LIN {X 0,Y 572.946,Z 406.186,A -85,B 0,C 180,E1 -2251.405,E2 -2251.405} C_VEL
LIN {X 0,Y 572.959,Z 403.811,A -85,B 0,C 180,E1 -2252.812,E2 -2252.812} C_VEL
LIN {X 0,Y 573.014,Z 400.897,A -85,B 0,C 180,E1 -2253.868,E2 -2253.868} C_VEL
LIN {X 0,Y 572.963,Z 396.95,A -85,B 0,C 180,E1 -2254.925,E2 -2254.925} C_VEL
LIN {X 0,Y 573.093,Z 391.869,A -85,B 0,C 180,E1 -2255.983,E2 -2255.983} C_VEL
LIN {X 0,Y 573.103,Z 385.471,A -85,B 0,C 180,E1 -2257.043,E2 -2257.043} C_VEL
LIN {X 0,Y 573.177,Z 377.482,A -85,B 0,C 180,E1 -2258.106,E2 -2258.106} C_VEL
LIN {X 0,Y 573.253,Z 369.34,A -85,B 0,C 180,E1 -2258.992,E2 -2258.992} C_VEL
LIN {X 0,Y 573.349,Z 359.406,A -85,B 0,C 180,E1 -2259.881,E2 -2259.881} C_VEL
LIN {X 0,Y 573.523,Z 348.194,A -85,B 0,C 180,E1 -2260.68,E2 -2260.68} C_VEL
LIN {X 0,Y 573.627,Z 337.186,A -85,B 0,C 180,E1 -2261.304,E2 -2261.304} C_VEL
LIN {X 0,Y 573.705,Z 324.996,A -85,B 0,C 180,E1 -2261.84,E2 -2261.84} C_VEL
LIN {X 0,Y 573.851,Z 312.2,A -85,B 0,C 180,E1 -2262.241,E2 -2262.241} C_VEL
LIN {X 0,Y 573.908,Z 298.642,A -85,B 0,C 180,E1 -2262.509,E2 -2262.509} C_VEL
LIN {X 0,Y 573.923,Z 199.106,A -85,B 0,C 180,E1 -2263.765,E2 -2263.765} C_VEL
LIN {X 0,Y 573.375,Z 195.407,A -85,B 0,C 180,E1 -2263.85,E2 -2263.85} C_VEL
LIN {X 0,Y 573.472,Z 178.674,A -85,B 0,C 180,E1 -2266.371,E2 -2266.371} C_VEL
LIN {X 0,Y 573.665,Z 161.996,A -85,B 0,C 180,E1 -2268.944,E2 -2268.944} C_VEL
LIN {X 0,Y 573.818,Z 145.276,A -85,B 0,C 180,E1 -2271.557,E2 -2271.557} C_VEL
LIN {X 0,Y 573.241,Z 142.129,A -85,B 0,C 180,E1 -2272.123,E2 -2272.123} C_VEL
LIN {X 0,Y 573.219,Z 142.079,A -85,B 0,C 180,E1 -2274.867,E2 -2274.867} C_VEL
LIN {X 0,Y 573.259,Z 142.075,A -85,B 0,C 180,E1 -2277.765,E2 -2277.765} C_VEL
LIN {X 0,Y 573.227,Z 142.075,A -85,B 0,C 180,E1 -2280.176,E2 -2280.176} C_VEL
LIN {X 0,Y 573.246,Z 142.076,A -85,B 0,C 180,E1 -2282.644,E2 -2282.644} C_VEL
LIN {X 0,Y 573.2,Z 142.088,A -85,B 0,C 180,E1 -2285.187,E2 -2285.187} C_VEL
LIN {X 0,Y 573.223,Z 142.075,A -85,B 0,C 180,E1 -2287.807,E2 -2287.807} C_VEL
LIN {X 0,Y 573.238,Z 142.076,A -85,B 0,C 180,E1 -2290.524,E2 -2290.524} C_VEL
LIN {X 0,Y 573.229,Z 142.077,A -85,B 0,C 180,E1 -2293.667,E2 -2293.667} C_VEL
LIN {X 0,Y 573.223,Z 142.079,A -85,B 0,C 180,E1 -2296.639,E2 -2296.639} C_VEL
LIN {X 0,Y 573.236,Z 142.078,A -85,B 0,C 180,E1 -2299.474,E2 -2299.474} C_VEL
LIN {X 0,Y 573.224,Z 142.074,A -85,B 0,C 180,E1 -2302.191,E2 -2302.191} C_VEL
LIN {X 0,Y 573.23,Z 142.08,A -85,B 0,C 180,E1 -2305.227,E2 -2305.227} C_VEL
LIN {X 0,Y 573.227,Z 142.076,A -85,B 0,C 180,E1 -2308.184,E2 -2308.184} C_VEL
LIN {X 0,Y 573.246,Z 142.078,A -85,B 0,C 180,E1 -2310.633,E2 -2310.633} C_VEL
LIN {X 0,Y 573.238,Z 142.082,A -85,B 0,C 180,E1 -2313.023,E2 -2313.023} C_VEL
LIN {X 0,Y 573.26,Z 142.072,A -85,B 0,C 180,E1 -2315.365,E2 -2315.365} C_VEL
LIN {X 0,Y 573.215,Z 142.081,A -85,B 0,C 180,E1 -2318.419,E2 -2318.419} C_VEL
LIN {X 0,Y 573.265,Z 142.08,A -85,B 0,C 180,E1 -2320.728,E2 -2320.728} C_VEL
LIN {X 0,Y 573.234,Z 142.074,A -85,B 0,C 180,E1 -2323.621,E2 -2323.621} C_VEL
LIN {X 0,Y 573.251,Z 142.073,A -85,B 0,C 180,E1 -2325.806,E2 -2325.806} C_VEL
LIN {X 0,Y 573.277,Z 142.077,A -85,B 0,C 180,E1 -2328.731,E2 -2328.731} C_VEL
LIN {X 0,Y 573.239,Z 142.074,A -85,B 0,C 180,E1 -2331.54,E2 -2331.54} C_VEL
LIN {X 0,Y 573.219,Z 142.076,A -85,B 0,C 180,E1 -2333.665,E2 -2333.665} C_VEL
LIN {X 0,Y 573.201,Z 142.077,A -85,B 0,C 180,E1 -2335.781,E2 -2335.781} C_VEL
LIN {X 0,Y 573.284,Z 142.07,A -85,B 0,C 180,E1 -2337.892,E2 -2337.892} C_VEL
LIN {X 0,Y 573.329,Z 142.068,A -85,B 0,C 180,E1 -2340.702,E2 -2340.702} C_VEL
LIN {X 0,Y 573.215,Z 142.076,A -85,B 0,C 180,E1 -2343.515,E2 -2343.515} C_VEL
LIN {X 0,Y 573.27,Z 142.07,A -85,B 0,C 180,E1 -2345.628,E2 -2345.628} C_VEL
LIN {X 0,Y 573.275,Z 142.077,A -85,B 0,C 180,E1 -2348.46,E2 -2348.46} C_VEL
LIN {X 0,Y 573.265,Z 142.07,A -85,B 0,C 180,E1 -2351.312,E2 -2351.312} C_VEL
LIN {X 0,Y 573.267,Z 142.078,A -85,B 0,C 180,E1 -2354.425,E2 -2354.425} C_VEL
LIN {X 0,Y 573.246,Z 142.073,A -85,B 0,C 180,E1 -2357.112,E2 -2357.112} C_VEL
LIN {X 0,Y 573.244,Z 142.081,A -85,B 0,C 180,E1 -2360.077,E2 -2360.077} C_VEL
LIN {X 0,Y 573.236,Z 142.082,A -85,B 0,C 180,E1 -2362.338,E2 -2362.338} C_VEL
LIN {X 0,Y 573.239,Z 142.076,A -85,B 0,C 180,E1 -2364.409,E2 -2364.409} C_VEL
LIN {X 0,Y 572.612,Z 142.157,A -85,B 0,C 180,E1 -2364.995,E2 -2364.995} C_VEL
LIN {X 0,Y 569.767,Z 142.513,A -85,B 0,C 180,E1 -2365.947,E2 -2365.947} C_VEL
LIN {X 0,Y 567.337,Z 142.81,A -85,B 0,C 180,E1 -2366.713,E2 -2366.713} C_VEL
LIN {X 0,Y 566.287,Z 142.939,A -85,B 0,C 180,E1 -2367.304,E2 -2367.304} C_VEL
LIN {X 0,Y 566.2,Z 142.951,A -85,B 0,C 180,E1 -2367.504,E2 -2367.504} C_VEL
LIN {X 0,Y 566.194,Z 142.956,A -85,B 0,C 180,E1 -2369.769,E2 -2369.769} C_VEL
LIN {X 0,Y 566.195,Z 142.954,A -85,B 0,C 180,E1 -2372.431,E2 -2372.431} C_VEL
LIN {X 0,Y 566.192,Z 142.946,A -85,B 0,C 180,E1 -2374.994,E2 -2374.994} C_VEL
LIN {X 0,Y 566.188,Z 142.952,A -85,B 0,C 180,E1 -2377.462,E2 -2377.462} C_VEL
LIN {X 0,Y 566.217,Z 142.955,A -85,B 0,C 180,E1 -2380.199,E2 -2380.199} C_VEL
LIN {X 0,Y 566.193,Z 142.948,A -85,B 0,C 180,E1 -2383.055,E2 -2383.055} C_VEL
LIN {X 0,Y 566.188,Z 142.961,A -85,B 0,C 180,E1 -2386.05,E2 -2386.05} C_VEL
LIN {X 0,Y 566.173,Z 142.953,A -85,B 0,C 180,E1 -2388.862,E2 -2388.862} C_VEL
LIN {X 0,Y 566.178,Z 142.958,A -85,B 0,C 180,E1 -2391.638,E2 -2391.638} C_VEL
LIN {X 0,Y 566.189,Z 142.954,A -85,B 0,C 180,E1 -2394.311,E2 -2394.311} C_VEL
LIN {X 0,Y 566.217,Z 142.949,A -85,B 0,C 180,E1 -2396.899,E2 -2396.899} C_VEL
LIN {X 0,Y 566.177,Z 142.957,A -85,B 0,C 180,E1 -2399.408,E2 -2399.408} C_VEL
LIN {X 0,Y 566.192,Z 142.961,A -85,B 0,C 180,E1 -2401.857,E2 -2401.857} C_VEL
LIN {X 0,Y 566.212,Z 142.953,A -85,B 0,C 180,E1 -2404.252,E2 -2404.252} C_VEL
LIN {X 0,Y 566.169,Z 142.956,A -85,B 0,C 180,E1 -2406.72,E2 -2406.72} C_VEL
LIN {X 0,Y 566.278,Z 143.111,A -85,B 0,C 180,E1 -2408.93,E2 -2408.93} C_VEL
LIN {X 0,Y 566.742,Z 147.362,A -85,B 0,C 180,E1 -2409.683,E2 -2409.683} C_VEL
LIN {X 0,Y 566.501,Z 165.312,A -85,B 0,C 180,E1 -2412.679,E2 -2412.679} C_VEL
LIN {X 0,Y 566.335,Z 182.135,A -85,B 0,C 180,E1 -2415.456,E2 -2415.456} C_VEL
LIN {X 0,Y 566.321,Z 185.792,A -85,B 0,C 180,E1 -2416.019,E2 -2416.019} C_VEL
LIN {X 0,Y 566.859,Z 189.275,A -85,B 0,C 180,E1 -2416.107,E2 -2416.107} C_VEL
LIN {X 0,Y 567.118,Z 197.768,A -85,B 0,C 180,E1 -2416.222,E2 -2416.222} C_VEL
LIN {X 0,Y 566.991,Z 292.999,A -85,B 0,C 180,E1 -2417.45,E2 -2417.45} C_VEL
LIN {X 0,Y 566.897,Z 306.243,A -85,B 0,C 180,E1 -2417.766,E2 -2417.766} C_VEL
LIN {X 0,Y 566.748,Z 318.396,A -85,B 0,C 180,E1 -2418.194,E2 -2418.194} C_VEL
LIN {X 0,Y 566.644,Z 330.553,A -85,B 0,C 180,E1 -2418.776,E2 -2418.776} C_VEL
LIN {X 0,Y 566.452,Z 341.562,A -85,B 0,C 180,E1 -2419.456,E2 -2419.456} C_VEL
LIN {X 0,Y 566.325,Z 352.079,A -85,B 0,C 180,E1 -2420.266,E2 -2420.266} C_VEL
LIN {X 0,Y 566.221,Z 360.675,A -85,B 0,C 180,E1 -2421.075,E2 -2421.075} C_VEL
LIN {X 0,Y 566.112,Z 368.594,A -85,B 0,C 180,E1 -2421.972,E2 -2421.972} C_VEL
LIN {X 0,Y 566.049,Z 375.161,A -85,B 0,C 180,E1 -2422.868,E2 -2422.868} C_VEL
LIN {X 0,Y 566.003,Z 381.63,A -85,B 0,C 180,E1 -2423.942,E2 -2423.942} C_VEL
LIN {X 0,Y 565.877,Z 386.766,A -85,B 0,C 180,E1 -2425.013,E2 -2425.013} C_VEL
LIN {X 0,Y 565.926,Z 390.755,A -85,B 0,C 180,E1 -2426.084,E2 -2426.084} C_VEL
LIN {X 0,Y 565.877,Z 393.704,A -85,B 0,C 180,E1 -2427.153,E2 -2427.153} C_VEL
LIN {X 0,Y 565.84,Z 395.127,A -85,B 0,C 180,E1 -2427.865,E2 -2427.865} C_VEL
LIN {X 0,Y 565.841,Z 396.757,A -85,B 0,C 180,E1 -2429.289,E2 -2429.289} C_VEL
LIN {X 0,Y 565.839,Z 396.996,A -85,B 0,C 180,E1 -2430,E2 -2430} C_VEL
LIN {X 0,Y 565.841,Z 396.815,A -85,B 0,C 180,E1 -2430.712,E2 -2430.712} C_VEL
LIN {X 0,Y 565.841,Z 395.266,A -85,B 0,C 180,E1 -2432.136,E2 -2432.136} C_VEL
LIN {X 0,Y 565.878,Z 393.905,A -85,B 0,C 180,E1 -2432.848,E2 -2432.848} C_VEL
LIN {X 0,Y 565.927,Z 391.029,A -85,B 0,C 180,E1 -2433.917,E2 -2433.917} C_VEL
LIN {X 0,Y 565.878,Z 387.128,A -85,B 0,C 180,E1 -2434.988,E2 -2434.988} C_VEL
LIN {X 0,Y 565.99,Z 382.096,A -85,B 0,C 180,E1 -2436.059,E2 -2436.059} C_VEL
LIN {X 0,Y 566.031,Z 375.771,A -85,B 0,C 180,E1 -2437.133,E2 -2437.133} C_VEL
LIN {X 0,Y 566.128,Z 367.849,A -85,B 0,C 180,E1 -2438.208,E2 -2438.208} C_VEL
LIN {X 0,Y 566.249,Z 357.997,A -85,B 0,C 180,E1 -2439.285,E2 -2439.285} C_VEL
LIN {X 0,Y 566.419,Z 347.678,A -85,B 0,C 180,E1 -2440.184,E2 -2440.184} C_VEL
LIN {X 0,Y 566.52,Z 336.387,A -85,B 0,C 180,E1 -2440.973,E2 -2440.973} C_VEL
LIN {X 0,Y 566.689,Z 325.186,A -85,B 0,C 180,E1 -2441.592,E2 -2441.592} C_VEL
LIN {X 0,Y 566.801,Z 312.592,A -85,B 0,C 180,E1 -2442.119,E2 -2442.119} C_VEL
LIN {X 0,Y 566.906,Z 299.416,A -85,B 0,C 180,E1 -2442.507,E2 -2442.507} C_VEL
LIN {X 0,Y 566.994,Z 287.047,A -85,B 0,C 180,E1 -2442.733,E2 -2442.733} C_VEL
LIN {X 0,Y 566.959,Z 189.903,A -85,B 0,C 180,E1 -2443.972,E2 -2443.972} C_VEL
LIN {X 0,Y 566.336,Z 185.757,A -85,B 0,C 180,E1 -2444.073,E2 -2444.073} C_VEL
LIN {X 0,Y 566.458,Z 168.51,A -85,B 0,C 180,E1 -2446.882,E2 -2446.882} C_VEL
LIN {X 0,Y 566.71,Z 150.14,A -85,B 0,C 180,E1 -2449.94,E2 -2449.94} C_VEL
LIN {X 0,Y 566.499,Z 144.518,A -85,B 0,C 180,E1 -2450.896,E2 -2450.896} C_VEL
LIN {X 0,Y 566.233,Z 142.988,A -85,B 0,C 180,E1 -2451.215,E2 -2451.215} C_VEL
LIN {X 0,Y 566.198,Z 142.959,A -85,B 0,C 180,E1 -2454.18,E2 -2454.18} C_VEL
LIN {X 0,Y 566.21,Z 142.956,A -85,B 0,C 180,E1 -2456.659,E2 -2456.659} C_VEL
LIN {X 0,Y 566.203,Z 142.952,A -85,B 0,C 180,E1 -2459.671,E2 -2459.671} C_VEL
LIN {X 0,Y 566.205,Z 142.959,A -85,B 0,C 180,E1 -2462.429,E2 -2462.429} C_VEL
LIN {X 0,Y 566.199,Z 142.95,A -85,B 0,C 180,E1 -2464.992,E2 -2464.992} C_VEL
LIN {X 0,Y 566.195,Z 142.953,A -85,B 0,C 180,E1 -2467.46,E2 -2467.46} C_VEL
LIN {X 0,Y 566.205,Z 142.956,A -85,B 0,C 180,E1 -2470.199,E2 -2470.199} C_VEL
LIN {X 0,Y 566.198,Z 142.952,A -85,B 0,C 180,E1 -2473.054,E2 -2473.054} C_VEL
LIN {X 0,Y 566.192,Z 142.958,A -85,B 0,C 180,E1 -2476.048,E2 -2476.048} C_VEL
LIN {X 0,Y 566.218,Z 142.948,A -85,B 0,C 180,E1 -2479.212,E2 -2479.212} C_VEL
LIN {X 0,Y 566.181,Z 142.957,A -85,B 0,C 180,E1 -2481.636,E2 -2481.636} C_VEL
LIN {X 0,Y 566.191,Z 142.95,A -85,B 0,C 180,E1 -2484.31,E2 -2484.31} C_VEL
LIN {X 0,Y 566.215,Z 142.947,A -85,B 0,C 180,E1 -2486.897,E2 -2486.897} C_VEL
LIN {X 0,Y 566.174,Z 142.957,A -85,B 0,C 180,E1 -2489.407,E2 -2489.407} C_VEL
LIN {X 0,Y 566.223,Z 142.957,A -85,B 0,C 180,E1 -2491.858,E2 -2491.858} C_VEL
LIN {X 0,Y 566.23,Z 142.948,A -85,B 0,C 180,E1 -2495.039,E2 -2495.039} C_VEL
LIN {X 0,Y 566.186,Z 142.956,A -85,B 0,C 180,E1 -2498.137,E2 -2498.137} C_VEL
LIN {X 0,Y 566.223,Z 142.949,A -85,B 0,C 180,E1 -2500.613,E2 -2500.613} C_VEL
LIN {X 0,Y 566.211,Z 142.953,A -85,B 0,C 180,E1 -2503.412,E2 -2503.412} C_VEL
LIN {X 0,Y 566.188,Z 142.953,A -85,B 0,C 180,E1 -2506.359,E2 -2506.359} C_VEL
LIN {X 0,Y 566.227,Z 142.947,A -85,B 0,C 180,E1 -2508.675,E2 -2508.675} C_VEL
LIN {X 0,Y 566.223,Z 142.952,A -85,B 0,C 180,E1 -2511.434,E2 -2511.434} C_VEL
LIN {X 0,Y 566.243,Z 142.947,A -85,B 0,C 180,E1 -2514.301,E2 -2514.301} C_VEL
LIN {X 0,Y 566.268,Z 142.945,A -85,B 0,C 180,E1 -2517.154,E2 -2517.154} C_VEL
LIN {X 0,Y 566.273,Z 142.945,A -85,B 0,C 180,E1 -2520,E2 -2520} C_VEL
LIN {X 0,Y 566.262,Z 142.944,A -85,B 0,C 180,E1 -2522.846,E2 -2522.846} C_VEL
LIN {X 0,Y 566.248,Z 142.95,A -85,B 0,C 180,E1 -2525.698,E2 -2525.698} C_VEL
LIN {X 0,Y 566.19,Z 142.953,A -85,B 0,C 180,E1 -2528.566,E2 -2528.566} C_VEL
LIN {X 0,Y 566.233,Z 142.954,A -85,B 0,C 180,E1 -2531.454,E2 -2531.454} C_VEL
LIN {X 0,Y 566.221,Z 142.949,A -85,B 0,C 180,E1 -2534.505,E2 -2534.505} C_VEL
LIN {X 0,Y 566.19,Z 142.96,A -85,B 0,C 180,E1 -2537.332,E2 -2537.332} C_VEL
LIN {X 0,Y 566.198,Z 142.951,A -85,B 0,C 180,E1 -2540.338,E2 -2540.338} C_VEL
LIN {X 0,Y 566.163,Z 142.963,A -85,B 0,C 180,E1 -2543.282,E2 -2543.282} C_VEL
LIN {X 0,Y 566.2,Z 142.953,A -85,B 0,C 180,E1 -2545.75,E2 -2545.75} C_VEL
LIN {X 0,Y 566.196,Z 142.951,A -85,B 0,C 180,E1 -2548.203,E2 -2548.203} C_VEL
LIN {X 0,Y 566.179,Z 142.962,A -85,B 0,C 180,E1 -2551.076,E2 -2551.076} C_VEL
LIN {X 0,Y 566.192,Z 142.952,A -85,B 0,C 180,E1 -2553.732,E2 -2553.732} C_VEL
LIN {X 0,Y 566.194,Z 142.95,A -85,B 0,C 180,E1 -2556.571,E2 -2556.571} C_VEL
LIN {X 0,Y 566.208,Z 142.951,A -85,B 0,C 180,E1 -2559.686,E2 -2559.686} C_VEL
LIN {X 0,Y 566.189,Z 142.961,A -85,B 0,C 180,E1 -2562.917,E2 -2562.917} C_VEL
LIN {X 0,Y 566.189,Z 142.953,A -85,B 0,C 180,E1 -2566.05,E2 -2566.05} C_VEL
LIN {X 0,Y 566.199,Z 142.955,A -85,B 0,C 180,E1 -2569.215,E2 -2569.215} C_VEL
LIN {X 0,Y 566.18,Z 142.951,A -85,B 0,C 180,E1 -2571.637,E2 -2571.637} C_VEL
LIN {X 0,Y 566.148,Z 142.961,A -85,B 0,C 180,E1 -2574.307,E2 -2574.307} C_VEL
LIN {X 0,Y 566.208,Z 142.959,A -85,B 0,C 180,E1 -2576.898,E2 -2576.898} C_VEL
LIN {X 0,Y 566.168,Z 142.956,A -85,B 0,C 180,E1 -2579.407,E2 -2579.407} C_VEL
LIN {X 0,Y 566.188,Z 142.953,A -85,B 0,C 180,E1 -2581.856,E2 -2581.856} C_VEL
LIN {X 0,Y 566.195,Z 142.955,A -85,B 0,C 180,E1 -2584.25,E2 -2584.25} C_VEL
LIN {X 0,Y 566.169,Z 142.96,A -85,B 0,C 180,E1 -2587.368,E2 -2587.368} C_VEL
LIN {X 0,Y 566.232,Z 143.18,A -85,B 0,C 180,E1 -2587.804,E2 -2587.804} C_VEL
LIN {X 0,Y 566.877,Z 148.388,A -85,B 0,C 180,E1 -2588.674,E2 -2588.674} C_VEL
LIN {X 0,Y 566.632,Z 166.706,A -85,B 0,C 180,E1 -2591.562,E2 -2591.562} C_VEL
LIN {X 0,Y 566.402,Z 184.608,A -85,B 0,C 180,E1 -2594.343,E2 -2594.343} C_VEL
LIN {X 0,Y 566.363,Z 195.4,A -85,B 0,C 180,E1 -2595.974,E2 -2595.974} C_VEL
LIN {X 0,Y 567.029,Z 199.971,A -85,B 0,C 180,E1 -2596.075,E2 -2596.075} C_VEL
LIN {X 0,Y 566.995,Z 302.945,A -85,B 0,C 180,E1 -2597.404,E2 -2597.404} C_VEL
LIN {X 0,Y 566.891,Z 316.217,A -85,B 0,C 180,E1 -2597.72,E2 -2597.72} C_VEL
LIN {X 0,Y 566.729,Z 328.377,A -85,B 0,C 180,E1 -2598.148,E2 -2598.148} C_VEL
LIN {X 0,Y 566.627,Z 340.152,A -85,B 0,C 180,E1 -2598.708,E2 -2598.708} C_VEL
LIN {X 0,Y 566.45,Z 352.195,A -85,B 0,C 180,E1 -2599.455,E2 -2599.455} C_VEL
LIN {X 0,Y 566.325,Z 362.603,A -85,B 0,C 180,E1 -2600.265,E2 -2600.265} C_VEL
LIN {X 0,Y 566.207,Z 371.112,A -85,B 0,C 180,E1 -2601.074,E2 -2601.074} C_VEL
LIN {X 0,Y 566.112,Z 378.96,A -85,B 0,C 180,E1 -2601.972,E2 -2601.972} C_VEL
LIN {X 0,Y 566.004,Z 386.622,A -85,B 0,C 180,E1 -2603.046,E2 -2603.046} C_VEL
LIN {X 0,Y 566.004,Z 393.679,A -85,B 0,C 180,E1 -2604.299,E2 -2604.299} C_VEL
LIN {X 0,Y 565.933,Z 398.372,A -85,B 0,C 180,E1 -2605.37,E2 -2605.37} C_VEL
LIN {X 0,Y 565.927,Z 401.957,A -85,B 0,C 180,E1 -2606.44,E2 -2606.44} C_VEL
LIN {X 0,Y 565.878,Z 403.807,A -85,B 0,C 180,E1 -2607.152,E2 -2607.152} C_VEL
LIN {X 0,Y 565.846,Z 406.184,A -85,B 0,C 180,E1 -2608.576,E2 -2608.576} C_VEL
LIN {X 0,Y 565.839,Z 407,A -85,B 0,C 180,E1 -2610,E2 -2610} C_VEL
LIN {X 0,Y 565.846,Z 406.185,A -85,B 0,C 180,E1 -2611.423,E2 -2611.423} C_VEL
LIN {X 0,Y 565.878,Z 403.811,A -85,B 0,C 180,E1 -2612.847,E2 -2612.847} C_VEL
LIN {X 0,Y 565.926,Z 400.897,A -85,B 0,C 180,E1 -2613.916,E2 -2613.916} C_VEL
LIN {X 0,Y 565.878,Z 396.95,A -85,B 0,C 180,E1 -2614.987,E2 -2614.987} C_VEL
LIN {X 0,Y 566.004,Z 391.87,A -85,B 0,C 180,E1 -2616.058,E2 -2616.058} C_VEL
LIN {X 0,Y 566.04,Z 385.471,A -85,B 0,C 180,E1 -2617.132,E2 -2617.132} C_VEL
LIN {X 0,Y 566.133,Z 377.482,A -85,B 0,C 180,E1 -2618.207,E2 -2618.207} C_VEL
LIN {X 0,Y 566.228,Z 369.339,A -85,B 0,C 180,E1 -2619.105,E2 -2619.105} C_VEL
LIN {X 0,Y 566.35,Z 359.405,A -85,B 0,C 180,E1 -2620.004,E2 -2620.004} C_VEL
LIN {X 0,Y 566.544,Z 348.293,A -85,B 0,C 180,E1 -2620.807,E2 -2620.807} C_VEL
LIN {X 0,Y 566.659,Z 337.184,A -85,B 0,C 180,E1 -2621.445,E2 -2621.445} C_VEL
LIN {X 0,Y 566.745,Z 324.993,A -85,B 0,C 180,E1 -2621.987,E2 -2621.987} C_VEL
LIN {X 0,Y 566.913,Z 312.198,A -85,B 0,C 180,E1 -2622.393,E2 -2622.393} C_VEL
LIN {X 0,Y 566.977,Z 298.641,A -85,B 0,C 180,E1 -2622.664,E2 -2622.664} C_VEL
LIN {X 0,Y 567.038,Z 199.913,A -85,B 0,C 180,E1 -2623.925,E2 -2623.925} C_VEL
LIN {X 0,Y 566.37,Z 195.419,A -85,B 0,C 180,E1 -2624.025,E2 -2624.025} C_VEL
LIN {X 0,Y 566.454,Z 179.839,A -85,B 0,C 180,E1 -2626.394,E2 -2626.394} C_VEL
LIN {X 0,Y 566.636,Z 164.32,A -85,B 0,C 180,E1 -2628.812,E2 -2628.812} C_VEL
LIN {X 0,Y 566.892,Z 146.706,A -85,B 0,C 180,E1 -2631.595,E2 -2631.595} C_VEL
LIN {X 0,Y 566.2,Z 143.056,A -85,B 0,C 180,E1 -2632.245,E2 -2632.245} C_VEL
LIN {X 0,Y 566.176,Z 142.958,A -85,B 0,C 180,E1 -2635.02,E2 -2635.02} C_VEL
LIN {X 0,Y 566.185,Z 142.957,A -85,B 0,C 180,E1 -2637.339,E2 -2637.339} C_VEL
LIN {X 0,Y 566.168,Z 142.958,A -85,B 0,C 180,E1 -2639.77,E2 -2639.77} C_VEL
LIN {X 0,Y 566.196,Z 142.953,A -85,B 0,C 180,E1 -2642.428,E2 -2642.428} C_VEL
LIN {X 0,Y 566.173,Z 142.959,A -85,B 0,C 180,E1 -2644.988,E2 -2644.988} C_VEL
LIN {X 0,Y 566.186,Z 142.955,A -85,B 0,C 180,E1 -2647.46,E2 -2647.46} C_VEL
LIN {X 0,Y 566.202,Z 142.951,A -85,B 0,C 180,E1 -2650.198,E2 -2650.198} C_VEL
LIN {X 0,Y 566.186,Z 142.961,A -85,B 0,C 180,E1 -2653.054,E2 -2653.054} C_VEL
LIN {X 0,Y 566.186,Z 142.952,A -85,B 0,C 180,E1 -2656.048,E2 -2656.048} C_VEL
LIN {X 0,Y 566.194,Z 142.959,A -85,B 0,C 180,E1 -2659.214,E2 -2659.214} C_VEL
LIN {X 0,Y 566.175,Z 142.953,A -85,B 0,C 180,E1 -2661.636,E2 -2661.636} C_VEL
LIN {X 0,Y 566.163,Z 142.952,A -85,B 0,C 180,E1 -2664.308,E2 -2664.308} C_VEL
LIN {X 0,Y 566.193,Z 142.96,A -85,B 0,C 180,E1 -2666.896,E2 -2666.896} C_VEL
LIN {X 0,Y 566.161,Z 142.957,A -85,B 0,C 180,E1 -2669.406,E2 -2669.406} C_VEL
LIN {X 0,Y 566.2,Z 142.951,A -85,B 0,C 180,E1 -2671.857,E2 -2671.857} C_VEL
LIN {X 0,Y 566.195,Z 142.953,A -85,B 0,C 180,E1 -2674.25,E2 -2674.25} C_VEL
LIN {X 0,Y 566.159,Z 142.963,A -85,B 0,C 180,E1 -2676.718,E2 -2676.718} C_VEL
LIN {X 0,Y 566.2,Z 142.951,A -85,B 0,C 180,E1 -2679.662,E2 -2679.662} C_VEL
LIN {X 0,Y 566.185,Z 142.96,A -85,B 0,C 180,E1 -2682.668,E2 -2682.668} C_VEL
LIN {X 0,Y 566.214,Z 142.949,A -85,B 0,C 180,E1 -2685.626,E2 -2685.626} C_VEL
LIN {X 0,Y 566.265,Z 142.95,A -85,B 0,C 180,E1 -2688.652,E2 -2688.652} C_VEL
LIN {X 0,Y 566.191,Z 142.952,A -85,B 0,C 180,E1 -2691.434,E2 -2691.434} C_VEL
LIN {X 0,Y 566.245,Z 142.95,A -85,B 0,C 180,E1 -2694.302,E2 -2694.302} C_VEL
LIN {X 0,Y 566.256,Z 142.945,A -85,B 0,C 180,E1 -2697.866,E2 -2697.866} C_VEL
LIN {X 0,Y 566.297,Z 142.944,A -85,B 0,C 180,E1 -2700.711,E2 -2700.711} C_VEL
LIN {X 0,Y 566.266,Z 142.945,A -85,B 0,C 180,E1 -2702.846,E2 -2702.846} C_VEL
LIN {X 0,Y 566.239,Z 142.947,A -85,B 0,C 180,E1 -2705.699,E2 -2705.699} C_VEL
LIN {X 0,Y 566.219,Z 142.953,A -85,B 0,C 180,E1 -2708.566,E2 -2708.566} C_VEL
LIN {X 0,Y 566.231,Z 142.947,A -85,B 0,C 180,E1 -2711.455,E2 -2711.455} C_VEL
LIN {X 0,Y 566.22,Z 142.954,A -85,B 0,C 180,E1 -2714.507,E2 -2714.507} C_VEL
LIN {X 0,Y 566.187,Z 142.952,A -85,B 0,C 180,E1 -2717.332,E2 -2717.332} C_VEL
LIN {X 0,Y 566.207,Z 142.958,A -85,B 0,C 180,E1 -2720.338,E2 -2720.338} C_VEL
LIN {X 0,Y 566.181,Z 142.953,A -85,B 0,C 180,E1 -2723.404,E2 -2723.404} C_VEL
LIN {X 0,Y 566.199,Z 142.955,A -85,B 0,C 180,E1 -2725.75,E2 -2725.75} C_VEL
LIN {X 0,Y 566.2,Z 142.951,A -85,B 0,C 180,E1 -2727.504,E2 -2727.504} C_VEL
LIN {X 0,Y 565.525,Z 143.043,A -85,B 0,C 180,E1 -2728.098,E2 -2728.098} C_VEL
LIN {X 0,Y 562.657,Z 143.401,A -85,B 0,C 180,E1 -2729.061,E2 -2729.061} C_VEL
LIN {X 0,Y 560.242,Z 143.701,A -85,B 0,C 180,E1 -2729.837,E2 -2729.837} C_VEL
LIN {X 0,Y 559.212,Z 143.827,A -85,B 0,C 180,E1 -2730.435,E2 -2730.435} C_VEL
LIN {X 0,Y 559.132,Z 143.834,A -85,B 0,C 180,E1 -2730.638,E2 -2730.638} C_VEL
LIN {X 0,Y 559.153,Z 143.829,A -85,B 0,C 180,E1 -2733.576,E2 -2733.576} C_VEL
LIN {X 0,Y 559.152,Z 143.83,A -85,B 0,C 180,E1 -2736.448,E2 -2736.448} C_VEL
LIN {X 0,Y 559.165,Z 143.828,A -85,B 0,C 180,E1 -2738.935,E2 -2738.935} C_VEL
LIN {X 0,Y 559.183,Z 143.831,A -85,B 0,C 180,E1 -2741.769,E2 -2741.769} C_VEL
LIN {X 0,Y 559.132,Z 143.83,A -85,B 0,C 180,E1 -2744.74,E2 -2744.74} C_VEL
LIN {X 0,Y 559.168,Z 143.837,A -85,B 0,C 180,E1 -2747.864,E2 -2747.864} C_VEL
LIN {X 0,Y 559.167,Z 143.825,A -85,B 0,C 180,E1 -2751.067,E2 -2751.067} C_VEL
LIN {X 0,Y 559.154,Z 143.838,A -85,B 0,C 180,E1 -2753.792,E2 -2753.792} C_VEL
LIN {X 0,Y 559.159,Z 143.83,A -85,B 0,C 180,E1 -2756.426,E2 -2756.426} C_VEL
LIN {X 0,Y 559.152,Z 143.828,A -85,B 0,C 180,E1 -2758.982,E2 -2758.982} C_VEL
LIN {X 0,Y 559.166,Z 143.835,A -85,B 0,C 180,E1 -2761.62,E2 -2761.62} C_VEL
LIN {X 0,Y 559.176,Z 143.828,A -85,B 0,C 180,E1 -2764.703,E2 -2764.703} C_VEL
LIN {X 0,Y 559.14,Z 143.839,A -85,B 0,C 180,E1 -2767.848,E2 -2767.848} C_VEL
LIN {X 0,Y 559.24,Z 144.062,A -85,B 0,C 180,E1 -2768.821,E2 -2768.821} C_VEL
LIN {X 0,Y 559.784,Z 148.482,A -85,B 0,C 180,E1 -2769.612,E2 -2769.612} C_VEL
LIN {X 0,Y 559.495,Z 166.671,A -85,B 0,C 180,E1 -2772.682,E2 -2772.682} C_VEL
LIN {X 0,Y 559.304,Z 184.354,A -85,B 0,C 180,E1 -2775.631,E2 -2775.631} C_VEL
LIN {X 0,Y 559.312,Z 185.814,A -85,B 0,C 180,E1 -2775.841,E2 -2775.841} C_VEL
LIN {X 0,Y 560.114,Z 190.921,A -85,B 0,C 180,E1 -2775.957,E2 -2775.957} C_VEL
LIN {X 0,Y 560.087,Z 293.035,A -85,B 0,C 180,E1 -2777.293,E2 -2777.293} C_VEL
LIN {X 0,Y 559.952,Z 306.263,A -85,B 0,C 180,E1 -2777.612,E2 -2777.612} C_VEL
LIN {X 0,Y 559.8,Z 318.407,A -85,B 0,C 180,E1 -2778.046,E2 -2778.046} C_VEL
LIN {X 0,Y 559.682,Z 330.094,A -85,B 0,C 180,E1 -2778.608,E2 -2778.608} C_VEL
LIN {X 0,Y 559.474,Z 341.567,A -85,B 0,C 180,E1 -2779.323,E2 -2779.323} C_VEL
LIN {X 0,Y 559.307,Z 352.084,A -85,B 0,C 180,E1 -2780.143,E2 -2780.143} C_VEL
LIN {X 0,Y 559.196,Z 360.68,A -85,B 0,C 180,E1 -2780.962,E2 -2780.962} C_VEL
LIN {X 0,Y 559.05,Z 368.599,A -85,B 0,C 180,E1 -2781.87,E2 -2781.87} C_VEL
LIN {X 0,Y 558.971,Z 376.46,A -85,B 0,C 180,E1 -2782.977,E2 -2782.977} C_VEL
LIN {X 0,Y 558.936,Z 383.456,A -85,B 0,C 180,E1 -2784.227,E2 -2784.227} C_VEL
LIN {X 0,Y 558.826,Z 388.196,A -85,B 0,C 180,E1 -2785.311,E2 -2785.311} C_VEL
LIN {X 0,Y 558.836,Z 391.829,A -85,B 0,C 180,E1 -2786.395,E2 -2786.395} C_VEL
LIN {X 0,Y 558.799,Z 393.706,A -85,B 0,C 180,E1 -2787.117,E2 -2787.117} C_VEL
LIN {X 0,Y 558.746,Z 395.127,A -85,B 0,C 180,E1 -2787.838,E2 -2787.838} C_VEL
LIN {X 0,Y 558.741,Z 396.757,A -85,B 0,C 180,E1 -2789.28,E2 -2789.28} C_VEL
LIN {X 0,Y 558.74,Z 396.996,A -85,B 0,C 180,E1 -2790,E2 -2790} C_VEL
LIN {X 0,Y 558.741,Z 396.815,A -85,B 0,C 180,E1 -2790.721,E2 -2790.721} C_VEL
LIN {X 0,Y 558.747,Z 395.264,A -85,B 0,C 180,E1 -2792.163,E2 -2792.163} C_VEL
LIN {X 0,Y 558.8,Z 393.903,A -85,B 0,C 180,E1 -2792.884,E2 -2792.884} C_VEL
LIN {X 0,Y 558.844,Z 391.027,A -85,B 0,C 180,E1 -2793.966,E2 -2793.966} C_VEL
LIN {X 0,Y 558.798,Z 387.126,A -85,B 0,C 180,E1 -2795.051,E2 -2795.051} C_VEL
LIN {X 0,Y 558.91,Z 382.094,A -85,B 0,C 180,E1 -2796.136,E2 -2796.136} C_VEL
LIN {X 0,Y 558.973,Z 375.767,A -85,B 0,C 180,E1 -2797.223,E2 -2797.223} C_VEL
LIN {X 0,Y 559.091,Z 367.844,A -85,B 0,C 180,E1 -2798.312,E2 -2798.312} C_VEL
LIN {X 0,Y 559.224,Z 357.99,A -85,B 0,C 180,E1 -2799.403,E2 -2799.403} C_VEL
LIN {X 0,Y 559.41,Z 347.668,A -85,B 0,C 180,E1 -2800.313,E2 -2800.313} C_VEL
LIN {X 0,Y 559.528,Z 336.697,A -85,B 0,C 180,E1 -2801.091,E2 -2801.091} C_VEL
LIN {X 0,Y 559.726,Z 325.174,A -85,B 0,C 180,E1 -2801.738,E2 -2801.738} C_VEL
LIN {X 0,Y 559.855,Z 312.575,A -85,B 0,C 180,E1 -2802.271,E2 -2802.271} C_VEL
LIN {X 0,Y 559.985,Z 299.398,A -85,B 0,C 180,E1 -2802.664,E2 -2802.664} C_VEL
LIN {X 0,Y 560.08,Z 287.014,A -85,B 0,C 180,E1 -2802.893,E2 -2802.893} C_VEL
LIN {X 0,Y 560.093,Z 190.667,A -85,B 0,C 180,E1 -2804.137,E2 -2804.137} C_VEL
LIN {X 0,Y 559.356,Z 186.125,A -85,B 0,C 180,E1 -2804.229,E2 -2804.229} C_VEL
LIN {X 0,Y 559.29,Z 184.891,A -85,B 0,C 180,E1 -2804.37,E2 -2804.37} C_VEL
LIN {X 0,Y 559.471,Z 168.832,A -85,B 0,C 180,E1 -2807.048,E2 -2807.048} C_VEL
LIN {X 0,Y 559.743,Z 151.249,A -85,B 0,C 180,E1 -2810.007,E2 -2810.007} C_VEL
LIN {X 0,Y 559.679,Z 146.751,A -85,B 0,C 180,E1 -2810.777,E2 -2810.777} C_VEL
LIN {X 0,Y 559.186,Z 143.901,A -85,B 0,C 180,E1 -2811.327,E2 -2811.327} C_VEL
LIN {X 0,Y 559.158,Z 143.837,A -85,B 0,C 180,E1 -2814.505,E2 -2814.505} C_VEL
LIN {X 0,Y 559.17,Z 143.83,A -85,B 0,C 180,E1 -2816.902,E2 -2816.902} C_VEL
LIN {X 0,Y 559.148,Z 143.833,A -85,B 0,C 180,E1 -2819.857,E2 -2819.857} C_VEL
LIN {X 0,Y 559.157,Z 143.832,A -85,B 0,C 180,E1 -2822.715,E2 -2822.715} C_VEL
LIN {X 0,Y 559.144,Z 143.828,A -85,B 0,C 180,E1 -2825.322,E2 -2825.322} C_VEL
LIN {X 0,Y 559.13,Z 143.839,A -85,B 0,C 180,E1 -2828.017,E2 -2828.017} C_VEL
LIN {X 0,Y 559.156,Z 143.828,A -85,B 0,C 180,E1 -2830.812,E2 -2830.812} C_VEL
LIN {X 0,Y 559.144,Z 143.83,A -85,B 0,C 180,E1 -2833.196,E2 -2833.196} C_VEL
LIN {X 0,Y 559.135,Z 143.834,A -85,B 0,C 180,E1 -2836.265,E2 -2836.265} C_VEL
LIN {X 0,Y 559.171,Z 143.826,A -85,B 0,C 180,E1 -2839.189,E2 -2839.189} C_VEL
LIN {X 0,Y 559.128,Z 143.841,A -85,B 0,C 180,E1 -2841.982,E2 -2841.982} C_VEL
LIN {X 0,Y 559.142,Z 143.823,A -85,B 0,C 180,E1 -2844.784,E2 -2844.784} C_VEL
LIN {X 0,Y 559.151,Z 143.828,A -85,B 0,C 180,E1 -2847.364,E2 -2847.364} C_VEL
LIN {X 0,Y 559.142,Z 143.836,A -85,B 0,C 180,E1 -2850.142,E2 -2850.142} C_VEL
LIN {X 0,Y 559.164,Z 143.827,A -85,B 0,C 180,E1 -2853.097,E2 -2853.097} C_VEL
LIN {X 0,Y 559.149,Z 143.834,A -85,B 0,C 180,E1 -2855.494,E2 -2855.494} C_VEL
LIN {X 0,Y 559.164,Z 143.826,A -85,B 0,C 180,E1 -2858.623,E2 -2858.623} C_VEL
LIN {X 0,Y 559.155,Z 143.829,A -85,B 0,C 180,E1 -2860.926,E2 -2860.926} C_VEL
LIN {X 0,Y 559.16,Z 143.832,A -85,B 0,C 180,E1 -2863.948,E2 -2863.948} C_VEL
LIN {X 0,Y 559.163,Z 143.83,A -85,B 0,C 180,E1 -2866.184,E2 -2866.184} C_VEL
LIN {X 0,Y 559.187,Z 143.826,A -85,B 0,C 180,E1 -2869.133,E2 -2869.133} C_VEL
LIN {X 0,Y 559.196,Z 143.826,A -85,B 0,C 180,E1 -2872.053,E2 -2872.053} C_VEL
LIN {X 0,Y 559.246,Z 143.818,A -85,B 0,C 180,E1 -2874.953,E2 -2874.953} C_VEL
LIN {X 0,Y 559.236,Z 143.822,A -85,B 0,C 180,E1 -2877.839,E2 -2877.839} C_VEL
LIN {X 0,Y 559.262,Z 143.816,A -85,B 0,C 180,E1 -2880.72,E2 -2880.72} C_VEL
LIN {X 0,Y 559.229,Z 143.821,A -85,B 0,C 180,E1 -2882.881,E2 -2882.881} C_VEL
LIN {X 0,Y 559.216,Z 143.825,A -85,B 0,C 180,E1 -2885.77,E2 -2885.77} C_VEL
LIN {X 0,Y 559.156,Z 143.829,A -85,B 0,C 180,E1 -2888.675,E2 -2888.675} C_VEL
LIN {X 0,Y 559.197,Z 143.828,A -85,B 0,C 180,E1 -2891.601,E2 -2891.601} C_VEL
LIN {X 0,Y 559.192,Z 143.825,A -85,B 0,C 180,E1 -2894.596,E2 -2894.596} C_VEL
LIN {X 0,Y 559.133,Z 143.835,A -85,B 0,C 180,E1 -2897.558,E2 -2897.558} C_VEL
LIN {X 0,Y 559.157,Z 143.83,A -85,B 0,C 180,E1 -2899.838,E2 -2899.838} C_VEL
LIN {X 0,Y 559.132,Z 143.831,A -85,B 0,C 180,E1 -2902.153,E2 -2902.153} C_VEL
LIN {X 0,Y 559.168,Z 143.835,A -85,B 0,C 180,E1 -2905.299,E2 -2905.299} C_VEL
LIN {X 0,Y 559.15,Z 143.831,A -85,B 0,C 180,E1 -2907.714,E2 -2907.714} C_VEL
LIN {X 0,Y 559.141,Z 143.83,A -85,B 0,C 180,E1 -2910.184,E2 -2910.184} C_VEL
LIN {X 0,Y 559.146,Z 143.834,A -85,B 0,C 180,E1 -2912.716,E2 -2912.716} C_VEL
LIN {X 0,Y 559.122,Z 143.833,A -85,B 0,C 180,E1 -2915.325,E2 -2915.325} C_VEL
LIN {X 0,Y 559.125,Z 143.829,A -85,B 0,C 180,E1 -2918.018,E2 -2918.018} C_VEL
LIN {X 0,Y 559.15,Z 143.836,A -85,B 0,C 180,E1 -2920.813,E2 -2920.813} C_VEL
LIN {X 0,Y 559.106,Z 143.835,A -85,B 0,C 180,E1 -2923.738,E2 -2923.738} C_VEL
LIN {X 0,Y 559.132,Z 143.833,A -85,B 0,C 180,E1 -2926.266,E2 -2926.266} C_VEL
LIN {X 0,Y 559.151,Z 143.834,A -85,B 0,C 180,E1 -2929.188,E2 -2929.188} C_VEL
LIN {X 0,Y 559.127,Z 143.829,A -85,B 0,C 180,E1 -2931.983,E2 -2931.983} C_VEL
LIN {X 0,Y 559.127,Z 143.841,A -85,B 0,C 180,E1 -2934.788,E2 -2934.788} C_VEL
LIN {X 0,Y 559.152,Z 143.832,A -85,B 0,C 180,E1 -2937.365,E2 -2937.365} C_VEL
LIN {X 0,Y 559.119,Z 143.835,A -85,B 0,C 180,E1 -2940.148,E2 -2940.148} C_VEL
LIN {X 0,Y 559.158,Z 143.831,A -85,B 0,C 180,E1 -2943.097,E2 -2943.097} C_VEL
LIN {X 0,Y 559.117,Z 143.833,A -85,B 0,C 180,E1 -2945.493,E2 -2945.493} C_VEL
LIN {X 0,Y 559.192,Z 144.03,A -85,B 0,C 180,E1 -2947.655,E2 -2947.655} C_VEL
LIN {X 0,Y 559.907,Z 148.304,A -85,B 0,C 180,E1 -2948.391,E2 -2948.391} C_VEL
LIN {X 0,Y 559.681,Z 164.253,A -85,B 0,C 180,E1 -2950.945,E2 -2950.945} C_VEL
LIN {X 0,Y 559.478,Z 179.771,A -85,B 0,C 180,E1 -2953.395,E2 -2953.395} C_VEL
LIN {X 0,Y 559.366,Z 195.367,A -85,B 0,C 180,E1 -2955.795,E2 -2955.795} C_VEL
LIN {X 0,Y 560.16,Z 200.844,A -85,B 0,C 180,E1 -2955.913,E2 -2955.913} C_VEL
LIN {X 0,Y 560.086,Z 302.945,A -85,B 0,C 180,E1 -2957.246,E2 -2957.246} C_VEL
LIN {X 0,Y 559.935,Z 316.216,A -85,B 0,C 180,E1 -2957.565,E2 -2957.565} C_VEL
LIN {X 0,Y 559.776,Z 328.375,A -85,B 0,C 180,E1 -2957.999,E2 -2957.999} C_VEL
LIN {X 0,Y 559.669,Z 339.812,A -85,B 0,C 180,E1 -2958.547,E2 -2958.547} C_VEL
LIN {X 0,Y 559.481,Z 350.901,A -85,B 0,C 180,E1 -2959.231,E2 -2959.231} C_VEL
LIN {X 0,Y 559.317,Z 361.535,A -85,B 0,C 180,E1 -2960.051,E2 -2960.051} C_VEL
LIN {X 0,Y 559.162,Z 371.112,A -85,B 0,C 180,E1 -2960.961,E2 -2960.961} C_VEL
LIN {X 0,Y 559.05,Z 378.96,A -85,B 0,C 180,E1 -2961.869,E2 -2961.869} C_VEL
LIN {X 0,Y 558.944,Z 386.622,A -85,B 0,C 180,E1 -2962.958,E2 -2962.958} C_VEL
LIN {X 0,Y 558.935,Z 393.679,A -85,B 0,C 180,E1 -2964.227,E2 -2964.227} C_VEL
LIN {X 0,Y 558.826,Z 398.372,A -85,B 0,C 180,E1 -2965.311,E2 -2965.311} C_VEL
LIN {X 0,Y 558.836,Z 401.957,A -85,B 0,C 180,E1 -2966.395,E2 -2966.395} C_VEL
LIN {X 0,Y 558.799,Z 403.806,A -85,B 0,C 180,E1 -2967.116,E2 -2967.116} C_VEL
LIN {X 0,Y 558.745,Z 406.183,A -85,B 0,C 180,E1 -2968.558,E2 -2968.558} C_VEL
LIN {X 0,Y 558.74,Z 407,A -85,B 0,C 180,E1 -2970,E2 -2970} C_VEL
LIN {X 0,Y 558.745,Z 406.185,A -85,B 0,C 180,E1 -2971.441,E2 -2971.441} C_VEL
LIN {X 0,Y 558.799,Z 403.811,A -85,B 0,C 180,E1 -2972.883,E2 -2972.883} C_VEL
LIN {X 0,Y 558.844,Z 400.897,A -85,B 0,C 180,E1 -2973.966,E2 -2973.966} C_VEL
LIN {X 0,Y 558.798,Z 396.95,A -85,B 0,C 180,E1 -2975.05,E2 -2975.05} C_VEL
LIN {X 0,Y 558.92,Z 391.87,A -85,B 0,C 180,E1 -2976.135,E2 -2976.135} C_VEL
LIN {X 0,Y 558.977,Z 385.47,A -85,B 0,C 180,E1 -2977.222,E2 -2977.222} C_VEL
LIN {X 0,Y 559.098,Z 377.481,A -85,B 0,C 180,E1 -2978.311,E2 -2978.311} C_VEL
LIN {X 0,Y 559.185,Z 369.338,A -85,B 0,C 180,E1 -2979.221,E2 -2979.221} C_VEL
LIN {X 0,Y 559.361,Z 359.404,A -85,B 0,C 180,E1 -2980.131,E2 -2980.131} C_VEL
LIN {X 0,Y 559.558,Z 348.371,A -85,B 0,C 180,E1 -2980.938,E2 -2980.938} C_VEL
LIN {X 0,Y 559.702,Z 336.149,A -85,B 0,C 180,E1 -2981.643,E2 -2981.643} C_VEL
LIN {X 0,Y 559.827,Z 323.785,A -85,B 0,C 180,E1 -2982.184,E2 -2982.184} C_VEL
LIN {X 0,Y 559.997,Z 310.368,A -85,B 0,C 180,E1 -2982.594,E2 -2982.594} C_VEL
LIN {X 0,Y 560.092,Z 297.126,A -85,B 0,C 180,E1 -2982.846,E2 -2982.846} C_VEL
LIN {X 0,Y 560.183,Z 200.781,A -85,B 0,C 180,E1 -2984.087,E2 -2984.087} C_VEL
LIN {X 0,Y 559.371,Z 195.386,A -85,B 0,C 180,E1 -2984.204,E2 -2984.204} C_VEL
LIN {X 0,Y 559.541,Z 176.828,A -85,B 0,C 180,E1 -2987.067,E2 -2987.067} C_VEL
LIN {X 0,Y 559.756,Z 159.482,A -85,B 0,C 180,E1 -2989.815,E2 -2989.815} C_VEL
LIN {X 0,Y 559.855,Z 147.574,A -85,B 0,C 180,E1 -2991.729,E2 -2991.729} C_VEL
LIN {X 0,Y 559.156,Z 143.867,A -85,B 0,C 180,E1 -2992.419,E2 -2992.419} C_VEL
LIN {X 0,Y 559.128,Z 143.841,A -85,B 0,C 180,E1 -2995.299,E2 -2995.299} C_VEL
LIN {X 0,Y 559.133,Z 143.835,A -85,B 0,C 180,E1 -2997.714,E2 -2997.714} C_VEL
LIN {X 0,Y 559.134,Z 143.831,A -85,B 0,C 180,E1 -3000.183,E2 -3000.183} C_VEL
LIN {X 0,Y 559.149,Z 143.833,A -85,B 0,C 180,E1 -3002.714,E2 -3002.714} C_VEL
LIN {X 0,Y 559.118,Z 143.842,A -85,B 0,C 180,E1 -3005.323,E2 -3005.323} C_VEL
LIN {X 0,Y 559.124,Z 143.829,A -85,B 0,C 180,E1 -3008.017,E2 -3008.017} C_VEL
LIN {X 0,Y 559.147,Z 143.834,A -85,B 0,C 180,E1 -3010.812,E2 -3010.812} C_VEL
LIN {X 0,Y 559.129,Z 143.833,A -85,B 0,C 180,E1 -3013.733,E2 -3013.733} C_VEL
LIN {X 0,Y 559.135,Z 143.836,A -85,B 0,C 180,E1 -3016.803,E2 -3016.803} C_VEL
LIN {X 0,Y 559.146,Z 143.837,A -85,B 0,C 180,E1 -3019.187,E2 -3019.187} C_VEL
LIN {X 0,Y 559.122,Z 143.829,A -85,B 0,C 180,E1 -3021.981,E2 -3021.981} C_VEL
LIN {X 0,Y 559.13,Z 143.833,A -85,B 0,C 180,E1 -3024.785,E2 -3024.785} C_VEL
LIN {X 0,Y 559.143,Z 143.834,A -85,B 0,C 180,E1 -3027.364,E2 -3027.364} C_VEL
LIN {X 0,Y 559.131,Z 143.831,A -85,B 0,C 180,E1 -3030.143,E2 -3030.143} C_VEL
LIN {X 0,Y 559.158,Z 143.833,A -85,B 0,C 180,E1 -3033.172,E2 -3033.172} C_VEL
LIN {X 0,Y 559.142,Z 143.829,A -85,B 0,C 180,E1 -3035.494,E2 -3035.494} C_VEL
LIN {X 0,Y 559.158,Z 143.835,A -85,B 0,C 180,E1 -3038.623,E2 -3038.623} C_VEL
LIN {X 0,Y 559.154,Z 143.834,A -85,B 0,C 180,E1 -3040.926,E2 -3040.926} C_VEL
LIN {X 0,Y 559.151,Z 143.829,A -85,B 0,C 180,E1 -3043.947,E2 -3043.947} C_VEL
LIN {X 0,Y 559.154,Z 143.831,A -85,B 0,C 180,E1 -3046.184,E2 -3046.184} C_VEL
LIN {X 0,Y 559.226,Z 143.821,A -85,B 0,C 180,E1 -3049.134,E2 -3049.134} C_VEL
LIN {X 0,Y 559.182,Z 143.827,A -85,B 0,C 180,E1 -3052.053,E2 -3052.053} C_VEL
LIN {X 0,Y 559.239,Z 143.819,A -85,B 0,C 180,E1 -3054.953,E2 -3054.953} C_VEL
LIN {X 0,Y 559.229,Z 143.82,A -85,B 0,C 180,E1 -3057.839,E2 -3057.839} C_VEL
LIN {X 0,Y 559.266,Z 143.819,A -85,B 0,C 180,E1 -3060.72,E2 -3060.72} C_VEL
LIN {X 0,Y 559.231,Z 143.821,A -85,B 0,C 180,E1 -3062.881,E2 -3062.881} C_VEL
LIN {X 0,Y 559.209,Z 143.823,A -85,B 0,C 180,E1 -3065.77,E2 -3065.77} C_VEL
LIN {X 0,Y 559.178,Z 143.828,A -85,B 0,C 180,E1 -3068.675,E2 -3068.675} C_VEL
LIN {X 0,Y 559.193,Z 143.824,A -85,B 0,C 180,E1 -3071.601,E2 -3071.601} C_VEL
LIN {X 0,Y 559.186,Z 143.828,A -85,B 0,C 180,E1 -3074.596,E2 -3074.596} C_VEL
LIN {X 0,Y 559.147,Z 143.83,A -85,B 0,C 180,E1 -3077.557,E2 -3077.557} C_VEL
LIN {X 0,Y 559.163,Z 143.831,A -85,B 0,C 180,E1 -3079.838,E2 -3079.838} C_VEL
LIN {X 0,Y 559.136,Z 143.838,A -85,B 0,C 180,E1 -3082.153,E2 -3082.153} C_VEL
LIN {X 0,Y 559.167,Z 143.827,A -85,B 0,C 180,E1 -3085.188,E2 -3085.188} C_VEL
LIN {X 0,Y 559.181,Z 143.827,A -85,B 0,C 180,E1 -3087.712,E2 -3087.712} C_VEL
LIN {X 0,Y 559.132,Z 143.834,A -85,B 0,C 180,E1 -3090.638,E2 -3090.638} C_VEL
LIN {X 0,Y 558.472,Z 143.915,A -85,B 0,C 180,E1 -3091.24,E2 -3091.24} C_VEL
LIN {X 0,Y 555.607,Z 144.276,A -85,B 0,C 180,E1 -3092.216,E2 -3092.216} C_VEL
LIN {X 0,Y 553.193,Z 144.572,A -85,B 0,C 180,E1 -3093.001,E2 -3093.001} C_VEL
LIN {X 0,Y 552.175,Z 144.698,A -85,B 0,C 180,E1 -3093.608,E2 -3093.608} C_VEL
LIN {X 0,Y 552.102,Z 144.707,A -85,B 0,C 180,E1 -3093.813,E2 -3093.813} C_VEL
LIN {X 0,Y 552.101,Z 144.706,A -85,B 0,C 180,E1 -3096.748,E2 -3096.748} C_VEL
LIN {X 0,Y 552.122,Z 144.708,A -85,B 0,C 180,E1 -3099.528,E2 -3099.528} C_VEL
LIN {X 0,Y 552.124,Z 144.703,A -85,B 0,C 180,E1 -3102.426,E2 -3102.426} C_VEL
LIN {X 0,Y 552.089,Z 144.711,A -85,B 0,C 180,E1 -3105.564,E2 -3105.564} C_VEL
LIN {X 0,Y 552.124,Z 144.704,A -85,B 0,C 180,E1 -3108.556,E2 -3108.556} C_VEL
LIN {X 0,Y 552.111,Z 144.707,A -85,B 0,C 180,E1 -3111.412,E2 -3111.412} C_VEL
LIN {X 0,Y 552.097,Z 144.71,A -85,B 0,C 180,E1 -3114.159,E2 -3114.159} C_VEL
LIN {X 0,Y 552.112,Z 144.707,A -85,B 0,C 180,E1 -3116.815,E2 -3116.815} C_VEL
LIN {X 0,Y 552.099,Z 144.71,A -85,B 0,C 180,E1 -3119.392,E2 -3119.392} C_VEL
LIN {X 0,Y 552.101,Z 144.716,A -85,B 0,C 180,E1 -3121.902,E2 -3121.902} C_VEL
LIN {X 0,Y 552.155,Z 144.703,A -85,B 0,C 180,E1 -3124.651,E2 -3124.651} C_VEL
LIN {X 0,Y 552.091,Z 144.718,A -85,B 0,C 180,E1 -3127.55,E2 -3127.55} C_VEL
LIN {X 0,Y 552.164,Z 144.919,A -85,B 0,C 180,E1 -3128.683,E2 -3128.683} C_VEL
LIN {X 0,Y 552.815,Z 149.606,A -85,B 0,C 180,E1 -3129.537,E2 -3129.537} C_VEL
LIN {X 0,Y 552.494,Z 168.006,A -85,B 0,C 180,E1 -3132.68,E2 -3132.68} C_VEL
LIN {X 0,Y 552.296,Z 185.669,A -85,B 0,C 180,E1 -3135.64,E2 -3135.64} C_VEL
LIN {X 0,Y 552.472,Z 187.115,A -85,B 0,C 180,E1 -3135.706,E2 -3135.706} C_VEL
LIN {X 0,Y 553.374,Z 193.679,A -85,B 0,C 180,E1 -3135.817,E2 -3135.817} C_VEL
LIN {X 0,Y 553.189,Z 293.129,A -85,B 0,C 180,E1 -3137.131,E2 -3137.131} C_VEL
LIN {X 0,Y 553.014,Z 306.347,A -85,B 0,C 180,E1 -3137.454,E2 -3137.454} C_VEL
LIN {X 0,Y 552.853,Z 318.473,A -85,B 0,C 180,E1 -3137.893,E2 -3137.893} C_VEL
LIN {X 0,Y 552.717,Z 329.891,A -85,B 0,C 180,E1 -3138.447,E2 -3138.447} C_VEL
LIN {X 0,Y 552.496,Z 341.616,A -85,B 0,C 180,E1 -3139.186,E2 -3139.186} C_VEL
LIN {X 0,Y 552.305,Z 352.119,A -85,B 0,C 180,E1 -3140.016,E2 -3140.016} C_VEL
LIN {X 0,Y 552.152,Z 360.704,A -85,B 0,C 180,E1 -3140.846,E2 -3140.846} C_VEL
LIN {X 0,Y 552.007,Z 368.611,A -85,B 0,C 180,E1 -3141.766,E2 -3141.766} C_VEL
LIN {X 0,Y 551.894,Z 376.463,A -85,B 0,C 180,E1 -3142.887,E2 -3142.887} C_VEL
LIN {X 0,Y 551.868,Z 383.459,A -85,B 0,C 180,E1 -3144.153,E2 -3144.153} C_VEL
LIN {X 0,Y 551.725,Z 388.198,A -85,B 0,C 180,E1 -3145.251,E2 -3145.251} C_VEL
LIN {X 0,Y 551.75,Z 391.83,A -85,B 0,C 180,E1 -3146.349,E2 -3146.349} C_VEL
LIN {X 0,Y 551.723,Z 393.708,A -85,B 0,C 180,E1 -3147.08,E2 -3147.08} C_VEL
LIN {X 0,Y 551.657,Z 395.127,A -85,B 0,C 180,E1 -3147.81,E2 -3147.81} C_VEL
LIN {X 0,Y 551.642,Z 396.756,A -85,B 0,C 180,E1 -3149.27,E2 -3149.27} C_VEL
LIN {X 0,Y 551.641,Z 396.996,A -85,B 0,C 180,E1 -3150,E2 -3150} C_VEL
LIN {X 0,Y 551.641,Z 396.815,A -85,B 0,C 180,E1 -3150.73,E2 -3150.73} C_VEL
LIN {X 0,Y 551.657,Z 395.262,A -85,B 0,C 180,E1 -3152.191,E2 -3152.191} C_VEL
LIN {X 0,Y 551.724,Z 393.901,A -85,B 0,C 180,E1 -3152.921,E2 -3152.921} C_VEL
LIN {X 0,Y 551.764,Z 391.025,A -85,B 0,C 180,E1 -3154.017,E2 -3154.017} C_VEL
LIN {X 0,Y 551.723,Z 387.124,A -85,B 0,C 180,E1 -3155.116,E2 -3155.116} C_VEL
LIN {X 0,Y 551.811,Z 381.392,A -85,B 0,C 180,E1 -3156.349,E2 -3156.349} C_VEL
LIN {X 0,Y 551.925,Z 374.535,A -85,B 0,C 180,E1 -3157.5,E2 -3157.5} C_VEL
LIN {X 0,Y 552.063,Z 366.364,A -85,B 0,C 180,E1 -3158.603,E2 -3158.603} C_VEL
LIN {X 0,Y 552.197,Z 358.006,A -85,B 0,C 180,E1 -3159.524,E2 -3159.524} C_VEL
LIN {X 0,Y 552.397,Z 347.694,A -85,B 0,C 180,E1 -3160.445,E2 -3160.445} C_VEL
LIN {X 0,Y 552.575,Z 335.921,A -85,B 0,C 180,E1 -3161.286,E2 -3161.286} C_VEL
LIN {X 0,Y 552.774,Z 324.504,A -85,B 0,C 180,E1 -3161.923,E2 -3161.923} C_VEL
LIN {X 0,Y 552.932,Z 312.493,A -85,B 0,C 180,E1 -3162.432,E2 -3162.432} C_VEL
LIN {X 0,Y 553.058,Z 299.44,A -85,B 0,C 180,E1 -3162.826,E2 -3162.826} C_VEL
LIN {X 0,Y 553.188,Z 287.036,A -85,B 0,C 180,E1 -3163.056,E2 -3163.056} C_VEL
LIN {X 0,Y 553.264,Z 191.854,A -85,B 0,C 180,E1 -3164.3,E2 -3164.3} C_VEL
LIN {X 0,Y 552.313,Z 185.943,A -85,B 0,C 180,E1 -3164.427,E2 -3164.427} C_VEL
LIN {X 0,Y 552.473,Z 170.354,A -85,B 0,C 180,E1 -3167.013,E2 -3167.013} C_VEL
LIN {X 0,Y 552.784,Z 152.372,A -85,B 0,C 180,E1 -3170.076,E2 -3170.076} C_VEL
LIN {X 0,Y 552.7,Z 147.872,A -85,B 0,C 180,E1 -3170.857,E2 -3170.857} C_VEL
LIN {X 0,Y 552.141,Z 144.762,A -85,B 0,C 180,E1 -3171.466,E2 -3171.466} C_VEL
LIN {X 0,Y 552.104,Z 144.713,A -85,B 0,C 180,E1 -3174.038,E2 -3174.038} C_VEL
LIN {X 0,Y 552.122,Z 144.713,A -85,B 0,C 180,E1 -3176.456,E2 -3176.456} C_VEL
LIN {X 0,Y 552.11,Z 144.709,A -85,B 0,C 180,E1 -3178.928,E2 -3178.928} C_VEL
LIN {X 0,Y 552.112,Z 144.704,A -85,B 0,C 180,E1 -3181.475,E2 -3181.475} C_VEL
LIN {X 0,Y 552.134,Z 144.712,A -85,B 0,C 180,E1 -3184.17,E2 -3184.17} C_VEL
LIN {X 0,Y 552.109,Z 144.709,A -85,B 0,C 180,E1 -3186.746,E2 -3186.746} C_VEL
LIN {X 0,Y 552.127,Z 144.703,A -85,B 0,C 180,E1 -3189.527,E2 -3189.527} C_VEL
LIN {X 0,Y 552.129,Z 144.71,A -85,B 0,C 180,E1 -3192.425,E2 -3192.425} C_VEL
LIN {X 0,Y 552.093,Z 144.709,A -85,B 0,C 180,E1 -3195.562,E2 -3195.562} C_VEL
LIN {X 0,Y 552.133,Z 144.704,A -85,B 0,C 180,E1 -3198.676,E2 -3198.676} C_VEL
LIN {X 0,Y 552.113,Z 144.708,A -85,B 0,C 180,E1 -3201.41,E2 -3201.41} C_VEL
LIN {X 0,Y 552.098,Z 144.706,A -85,B 0,C 180,E1 -3204.157,E2 -3204.157} C_VEL
LIN {X 0,Y 552.11,Z 144.704,A -85,B 0,C 180,E1 -3206.814,E2 -3206.814} C_VEL
LIN {X 0,Y 552.096,Z 144.71,A -85,B 0,C 180,E1 -3209.39,E2 -3209.39} C_VEL
LIN {X 0,Y 552.12,Z 144.712,A -85,B 0,C 180,E1 -3211.902,E2 -3211.902} C_VEL
LIN {X 0,Y 552.131,Z 144.704,A -85,B 0,C 180,E1 -3214.653,E2 -3214.653} C_VEL
LIN {X 0,Y 552.085,Z 144.714,A -85,B 0,C 180,E1 -3217.549,E2 -3217.549} C_VEL
LIN {X 0,Y 552.137,Z 144.705,A -85,B 0,C 180,E1 -3220.374,E2 -3220.374} C_VEL
LIN {X 0,Y 552.149,Z 144.701,A -85,B 0,C 180,E1 -3222.977,E2 -3222.977} C_VEL
LIN {X 0,Y 552.127,Z 144.709,A -85,B 0,C 180,E1 -3226.004,E2 -3226.004} C_VEL
LIN {X 0,Y 552.154,Z 144.701,A -85,B 0,C 180,E1 -3228.993,E2 -3228.993} C_VEL
LIN {X 0,Y 552.15,Z 144.705,A -85,B 0,C 180,E1 -3231.951,E2 -3231.951} C_VEL
LIN {X 0,Y 552.22,Z 144.693,A -85,B 0,C 180,E1 -3234.889,E2 -3234.889} C_VEL
LIN {X 0,Y 552.209,Z 144.698,A -85,B 0,C 180,E1 -3237.812,E2 -3237.812} C_VEL
LIN {X 0,Y 552.233,Z 144.691,A -85,B 0,C 180,E1 -3240.729,E2 -3240.729} C_VEL
LIN {X 0,Y 552.196,Z 144.697,A -85,B 0,C 180,E1 -3242.918,E2 -3242.918} C_VEL
LIN {X 0,Y 552.186,Z 144.7,A -85,B 0,C 180,E1 -3245.844,E2 -3245.844} C_VEL
LIN {X 0,Y 552.132,Z 144.705,A -85,B 0,C 180,E1 -3248.786,E2 -3248.786} C_VEL
LIN {X 0,Y 552.154,Z 144.703,A -85,B 0,C 180,E1 -3251.751,E2 -3251.751} C_VEL
LIN {X 0,Y 552.128,Z 144.706,A -85,B 0,C 180,E1 -3254.749,E2 -3254.749} C_VEL
LIN {X 0,Y 552.091,Z 144.709,A -85,B 0,C 180,E1 -3257.789,E2 -3257.789} C_VEL
LIN {X 0,Y 552.118,Z 144.706,A -85,B 0,C 180,E1 -3260.102,E2 -3260.102} C_VEL
LIN {X 0,Y 552.084,Z 144.71,A -85,B 0,C 180,E1 -3262.451,E2 -3262.451} C_VEL
LIN {X 0,Y 552.13,Z 144.711,A -85,B 0,C 180,E1 -3265.347,E2 -3265.347} C_VEL
LIN {X 0,Y 552.09,Z 144.708,A -85,B 0,C 180,E1 -3268.1,E2 -3268.1} C_VEL
LIN {X 0,Y 552.091,Z 144.71,A -85,B 0,C 180,E1 -3270.61,E2 -3270.61} C_VEL
LIN {X 0,Y 552.101,Z 144.714,A -85,B 0,C 180,E1 -3273.187,E2 -3273.187} C_VEL
LIN {X 0,Y 552.08,Z 144.704,A -85,B 0,C 180,E1 -3275.844,E2 -3275.844} C_VEL
LIN {X 0,Y 552.115,Z 144.714,A -85,B 0,C 180,E1 -3279.061,E2 -3279.061} C_VEL
LIN {X 0,Y 552.115,Z 144.708,A -85,B 0,C 180,E1 -3281.447,E2 -3281.447} C_VEL
LIN {X 0,Y 552.071,Z 144.714,A -85,B 0,C 180,E1 -3284.53,E2 -3284.53} C_VEL
LIN {X 0,Y 552.105,Z 144.708,A -85,B 0,C 180,E1 -3287.588,E2 -3287.588} C_VEL
LIN {X 0,Y 552.128,Z 144.708,A -85,B 0,C 180,E1 -3290.473,E2 -3290.473} C_VEL
LIN {X 0,Y 552.097,Z 144.711,A -85,B 0,C 180,E1 -3293.319,E2 -3293.319} C_VEL
LIN {X 0,Y 552.123,Z 144.703,A -85,B 0,C 180,E1 -3295.939,E2 -3295.939} C_VEL
LIN {X 0,Y 552.12,Z 144.713,A -85,B 0,C 180,E1 -3298.541,E2 -3298.541} C_VEL
LIN {X 0,Y 552.102,Z 144.708,A -85,B 0,C 180,E1 -3301.443,E2 -3301.443} C_VEL
LIN {X 0,Y 552.104,Z 144.707,A -85,B 0,C 180,E1 -3303.543,E2 -3303.543} C_VEL
LIN {X 0,Y 552.09,Z 144.714,A -85,B 0,C 180,E1 -3306.758,E2 -3306.758} C_VEL
LIN {X 0,Y 552.139,Z 144.889,A -85,B 0,C 180,E1 -3307.502,E2 -3307.502} C_VEL
LIN {X 0,Y 552.949,Z 149.865,A -85,B 0,C 180,E1 -3308.371,E2 -3308.371} C_VEL
LIN {X 0,Y 552.702,Z 165.385,A -85,B 0,C 180,E1 -3310.887,E2 -3310.887} C_VEL
LIN {X 0,Y 552.491,Z 179.706,A -85,B 0,C 180,E1 -3313.178,E2 -3313.178} C_VEL
LIN {X 0,Y 552.358,Z 195.332,A -85,B 0,C 180,E1 -3315.613,E2 -3315.613} C_VEL
LIN {X 0,Y 553.43,Z 202.968,A -85,B 0,C 180,E1 -3315.767,E2 -3315.767} C_VEL
LIN {X 0,Y 553.151,Z 302.88,A -85,B 0,C 180,E1 -3317.083,E2 -3317.083} C_VEL
LIN {X 0,Y 553.023,Z 316.156,A -85,B 0,C 180,E1 -3317.407,E2 -3317.407} C_VEL
LIN {X 0,Y 552.827,Z 328.314,A -85,B 0,C 180,E1 -3317.845,E2 -3317.845} C_VEL
LIN {X 0,Y 552.69,Z 340.614,A -85,B 0,C 180,E1 -3318.449,E2 -3318.449} C_VEL
LIN {X 0,Y 552.479,Z 352.158,A -85,B 0,C 180,E1 -3319.185,E2 -3319.185} C_VEL
LIN {X 0,Y 552.276,Z 362.582,A -85,B 0,C 180,E1 -3320.015,E2 -3320.015} C_VEL
LIN {X 0,Y 552.126,Z 371.101,A -85,B 0,C 180,E1 -3320.845,E2 -3320.845} C_VEL
LIN {X 0,Y 552.013,Z 378.96,A -85,B 0,C 180,E1 -3321.765,E2 -3321.765} C_VEL
LIN {X 0,Y 551.889,Z 386.62,A -85,B 0,C 180,E1 -3322.868,E2 -3322.868} C_VEL
LIN {X 0,Y 551.867,Z 393.678,A -85,B 0,C 180,E1 -3324.152,E2 -3324.152} C_VEL
LIN {X 0,Y 551.725,Z 398.372,A -85,B 0,C 180,E1 -3325.25,E2 -3325.25} C_VEL
LIN {X 0,Y 551.75,Z 401.957,A -85,B 0,C 180,E1 -3326.348,E2 -3326.348} C_VEL
LIN {X 0,Y 551.723,Z 403.806,A -85,B 0,C 180,E1 -3327.079,E2 -3327.079} C_VEL
LIN {X 0,Y 551.645,Z 406.182,A -85,B 0,C 180,E1 -3328.54,E2 -3328.54} C_VEL
LIN {X 0,Y 551.64,Z 407,A -85,B 0,C 180,E1 -3330,E2 -3330} C_VEL
LIN {X 0,Y 551.645,Z 406.184,A -85,B 0,C 180,E1 -3331.46,E2 -3331.46} C_VEL
LIN {X 0,Y 551.723,Z 403.811,A -85,B 0,C 180,E1 -3332.92,E2 -3332.92} C_VEL
LIN {X 0,Y 551.764,Z 400.896,A -85,B 0,C 180,E1 -3334.017,E2 -3334.017} C_VEL
LIN {X 0,Y 551.723,Z 396.95,A -85,B 0,C 180,E1 -3335.115,E2 -3335.115} C_VEL
LIN {X 0,Y 551.823,Z 391.197,A -85,B 0,C 180,E1 -3336.34,E2 -3336.34} C_VEL
LIN {X 0,Y 551.926,Z 384.238,A -85,B 0,C 180,E1 -3337.499,E2 -3337.499} C_VEL
LIN {X 0,Y 552.082,Z 375.993,A -85,B 0,C 180,E1 -3338.602,E2 -3338.602} C_VEL
LIN {X 0,Y 552.224,Z 367.53,A -85,B 0,C 180,E1 -3339.523,E2 -3339.523} C_VEL
LIN {X 0,Y 552.422,Z 357.07,A -85,B 0,C 180,E1 -3340.444,E2 -3340.444} C_VEL
LIN {X 0,Y 552.6,Z 346.096,A -85,B 0,C 180,E1 -3341.223,E2 -3341.223} C_VEL
LIN {X 0,Y 552.752,Z 335.367,A -85,B 0,C 180,E1 -3341.83,E2 -3341.83} C_VEL
LIN {X 0,Y 552.882,Z 323.724,A -85,B 0,C 180,E1 -3342.339,E2 -3342.339} C_VEL
LIN {X 0,Y 553.091,Z 310.305,A -85,B 0,C 180,E1 -3342.754,E2 -3342.754} C_VEL
LIN {X 0,Y 553.179,Z 297.061,A -85,B 0,C 180,E1 -3343.009,E2 -3343.009} C_VEL
LIN {X 0,Y 553.375,Z 202.081,A -85,B 0,C 180,E1 -3344.247,E2 -3344.247} C_VEL
LIN {X 0,Y 552.359,Z 195.336,A -85,B 0,C 180,E1 -3344.387,E2 -3344.387} C_VEL
LIN {X 0,Y 552.549,Z 177.464,A -85,B 0,C 180,E1 -3347.178,E2 -3347.178} C_VEL
LIN {X 0,Y 552.863,Z 158.227,A -85,B 0,C 180,E1 -3350.267,E2 -3350.267} C_VEL
LIN {X 0,Y 552.821,Z 148.443,A -85,B 0,C 180,E1 -3351.867,E2 -3351.867} C_VEL
LIN {X 0,Y 552.119,Z 144.774,A -85,B 0,C 180,E1 -3352.548,E2 -3352.548} C_VEL
LIN {X 0,Y 552.083,Z 144.715,A -85,B 0,C 180,E1 -3355.646,E2 -3355.646} C_VEL
LIN {X 0,Y 552.084,Z 144.71,A -85,B 0,C 180,E1 -3358.099,E2 -3358.099} C_VEL
LIN {X 0,Y 552.091,Z 144.71,A -85,B 0,C 180,E1 -3360.609,E2 -3360.609} C_VEL
LIN {X 0,Y 552.109,Z 144.714,A -85,B 0,C 180,E1 -3363.185,E2 -3363.185} C_VEL
LIN {X 0,Y 552.07,Z 144.713,A -85,B 0,C 180,E1 -3365.843,E2 -3365.843} C_VEL
LIN {X 0,Y 552.111,Z 144.704,A -85,B 0,C 180,E1 -3368.588,E2 -3368.588} C_VEL
LIN {X 0,Y 552.102,Z 144.712,A -85,B 0,C 180,E1 -3371.446,E2 -3371.446} C_VEL
LIN {X 0,Y 552.083,Z 144.712,A -85,B 0,C 180,E1 -3374.53,E2 -3374.53} C_VEL
LIN {X 0,Y 552.121,Z 144.707,A -85,B 0,C 180,E1 -3377.584,E2 -3377.584} C_VEL
LIN {X 0,Y 552.12,Z 144.707,A -85,B 0,C 180,E1 -3380.472,E2 -3380.472} C_VEL
LIN {X 0,Y 552.097,Z 144.706,A -85,B 0,C 180,E1 -3383.316,E2 -3383.316} C_VEL
LIN {X 0,Y 552.095,Z 144.707,A -85,B 0,C 180,E1 -3385.937,E2 -3385.937} C_VEL
LIN {X 0,Y 552.108,Z 144.711,A -85,B 0,C 180,E1 -3388.54,E2 -3388.54} C_VEL
LIN {X 0,Y 552.093,Z 144.71,A -85,B 0,C 180,E1 -3391.441,E2 -3391.441} C_VEL
LIN {X 0,Y 552.116,Z 144.708,A -85,B 0,C 180,E1 -3394.355,E2 -3394.355} C_VEL
LIN {X 0,Y 552.085,Z 144.716,A -85,B 0,C 180,E1 -3396.757,E2 -3396.757} C_VEL
LIN {X 0,Y 552.107,Z 144.711,A -85,B 0,C 180,E1 -3399.119,E2 -3399.119} C_VEL
LIN {X 0,Y 552.11,Z 144.705,A -85,B 0,C 180,E1 -3401.444,E2 -3401.444} C_VEL
LIN {X 0,Y 552.101,Z 144.707,A -85,B 0,C 180,E1 -3403.737,E2 -3403.737} C_VEL
LIN {X 0,Y 552.119,Z 144.706,A -85,B 0,C 180,E1 -3406.004,E2 -3406.004} C_VEL
LIN {X 0,Y 552.185,Z 144.7,A -85,B 0,C 180,E1 -3408.994,E2 -3408.994} C_VEL
LIN {X 0,Y 552.136,Z 144.704,A -85,B 0,C 180,E1 -3411.951,E2 -3411.951} C_VEL
LIN {X 0,Y 552.214,Z 144.695,A -85,B 0,C 180,E1 -3414.889,E2 -3414.889} C_VEL
LIN {X 0,Y 552.202,Z 144.695,A -85,B 0,C 180,E1 -3417.812,E2 -3417.812} C_VEL
LIN {X 0,Y 552.235,Z 144.695,A -85,B 0,C 180,E1 -3420.729,E2 -3420.729} C_VEL
LIN {X 0,Y 552.196,Z 144.697,A -85,B 0,C 180,E1 -3422.918,E2 -3422.918} C_VEL
LIN {X 0,Y 552.18,Z 144.699,A -85,B 0,C 180,E1 -3425.844,E2 -3425.844} C_VEL
LIN {X 0,Y 552.148,Z 144.702,A -85,B 0,C 180,E1 -3428.786,E2 -3428.786} C_VEL
LIN {X 0,Y 552.15,Z 144.702,A -85,B 0,C 180,E1 -3431.751,E2 -3431.751} C_VEL
LIN {X 0,Y 552.123,Z 144.705,A -85,B 0,C 180,E1 -3434.749,E2 -3434.749} C_VEL
LIN {X 0,Y 552.098,Z 144.709,A -85,B 0,C 180,E1 -3437.789,E2 -3437.789} C_VEL
LIN {X 0,Y 552.122,Z 144.712,A -85,B 0,C 180,E1 -3440.102,E2 -3440.102} C_VEL
LIN {X 0,Y 552.089,Z 144.714,A -85,B 0,C 180,E1 -3442.451,E2 -3442.451} C_VEL
LIN {X 0,Y 552.143,Z 144.703,A -85,B 0,C 180,E1 -3445.351,E2 -3445.351} C_VEL
LIN {X 0,Y 552.115,Z 144.712,A -85,B 0,C 180,E1 -3448.098,E2 -3448.098} C_VEL
LIN {X 0,Y 552.094,Z 144.711,A -85,B 0,C 180,E1 -3450.634,E2 -3450.634} C_VEL
LIN {X 0,Y 552.105,Z 144.704,A -85,B 0,C 180,E1 -3453.187,E2 -3453.187} C_VEL
LIN {X 0,Y 552.102,Z 144.707,A -85,B 0,C 180,E1 -3453.813,E2 -3453.813} C_VEL
LIN {X 0,Y 551.47,Z 144.789,A -85,B 0,C 180,E1 -3454.422,E2 -3454.422} C_VEL
LIN {X 0,Y 548.647,Z 145.14,A -85,B 0,C 180,E1 -3455.41,E2 -3455.41} C_VEL
LIN {X 0,Y 546.225,Z 145.443,A -85,B 0,C 180,E1 -3456.205,E2 -3456.205} C_VEL
LIN {X 0,Y 545.155,Z 145.57,A -85,B 0,C 180,E1 -3456.819,E2 -3456.819} C_VEL
LIN {X 0,Y 545.053,Z 145.582,A -85,B 0,C 180,E1 -3457.027,E2 -3457.027} C_VEL
LIN {X 0,Y 545.064,Z 145.591,A -85,B 0,C 180,E1 -3460.143,E2 -3460.143} C_VEL
LIN {X 0,Y 545.055,Z 145.58,A -85,B 0,C 180,E1 -3462.698,E2 -3462.698} C_VEL
LIN {X 0,Y 545.03,Z 145.587,A -85,B 0,C 180,E1 -3465.171,E2 -3465.171} C_VEL
LIN {X 0,Y 545.075,Z 145.591,A -85,B 0,C 180,E1 -3467.898,E2 -3467.898} C_VEL
LIN {X 0,Y 545.073,Z 145.58,A -85,B 0,C 180,E1 -3470.819,E2 -3470.819} C_VEL
LIN {X 0,Y 545.045,Z 145.593,A -85,B 0,C 180,E1 -3473.621,E2 -3473.621} C_VEL
LIN {X 0,Y 545.063,Z 145.587,A -85,B 0,C 180,E1 -3476.329,E2 -3476.329} C_VEL
LIN {X 0,Y 545.063,Z 145.583,A -85,B 0,C 180,E1 -3478.953,E2 -3478.953} C_VEL
LIN {X 0,Y 545.098,Z 145.587,A -85,B 0,C 180,E1 -3481.509,E2 -3481.509} C_VEL
LIN {X 0,Y 545.094,Z 145.583,A -85,B 0,C 180,E1 -3484.492,E2 -3484.492} C_VEL
LIN {X 0,Y 545.036,Z 145.593,A -85,B 0,C 180,E1 -3487.243,E2 -3487.243} C_VEL
LIN {X 0,Y 545.124,Z 145.714,A -85,B 0,C 180,E1 -3488.522,E2 -3488.522} C_VEL
LIN {X 0,Y 545.847,Z 150.735,A -85,B 0,C 180,E1 -3489.461,E2 -3489.461} C_VEL
LIN {X 0,Y 545.522,Z 167.9,A -85,B 0,C 180,E1 -3492.431,E2 -3492.431} C_VEL
LIN {X 0,Y 545.311,Z 185.879,A -85,B 0,C 180,E1 -3495.464,E2 -3495.464} C_VEL
LIN {X 0,Y 546.023,Z 190.292,A -85,B 0,C 180,E1 -3495.575,E2 -3495.575} C_VEL
LIN {X 0,Y 546.497,Z 194.631,A -85,B 0,C 180,E1 -3495.646,E2 -3495.646} C_VEL
LIN {X 0,Y 546.294,Z 293.222,A -85,B 0,C 180,E1 -3496.966,E2 -3496.966} C_VEL
LIN {X 0,Y 546.105,Z 305.67,A -85,B 0,C 180,E1 -3497.269,E2 -3497.269} C_VEL
LIN {X 0,Y 545.907,Z 318.552,A -85,B 0,C 180,E1 -3497.736,E2 -3497.736} C_VEL
LIN {X 0,Y 545.734,Z 330.674,A -85,B 0,C 180,E1 -3498.339,E2 -3498.339} C_VEL
LIN {X 0,Y 545.516,Z 341.689,A -85,B 0,C 180,E1 -3499.046,E2 -3499.046} C_VEL
LIN {X 0,Y 545.296,Z 352.191,A -85,B 0,C 180,E1 -3499.887,E2 -3499.887} C_VEL
LIN {X 0,Y 545.121,Z 360.774,A -85,B 0,C 180,E1 -3500.727,E2 -3500.727} C_VEL
LIN {X 0,Y 544.975,Z 368.681,A -85,B 0,C 180,E1 -3501.659,E2 -3501.659} C_VEL
LIN {X 0,Y 544.829,Z 376.416,A -85,B 0,C 180,E1 -3502.775,E2 -3502.775} C_VEL
LIN {X 0,Y 544.8,Z 383.51,A -85,B 0,C 180,E1 -3504.077,E2 -3504.077} C_VEL
LIN {X 0,Y 544.629,Z 388.242,A -85,B 0,C 180,E1 -3505.189,E2 -3505.189} C_VEL
LIN {X 0,Y 544.669,Z 391.865,A -85,B 0,C 180,E1 -3506.301,E2 -3506.301} C_VEL
LIN {X 0,Y 544.65,Z 393.739,A -85,B 0,C 180,E1 -3507.042,E2 -3507.042} C_VEL
LIN {X 0,Y 544.571,Z 395.155,A -85,B 0,C 180,E1 -3507.782,E2 -3507.782} C_VEL
LIN {X 0,Y 544.542,Z 396.781,A -85,B 0,C 180,E1 -3509.261,E2 -3509.261} C_VEL
LIN {X 0,Y 544.542,Z 397.02,A -85,B 0,C 180,E1 -3510,E2 -3510} C_VEL
LIN {X 0,Y 544.542,Z 396.838,A -85,B 0,C 180,E1 -3510.74,E2 -3510.74} C_VEL
LIN {X 0,Y 544.572,Z 395.287,A -85,B 0,C 180,E1 -3512.219,E2 -3512.219} C_VEL
LIN {X 0,Y 544.651,Z 393.929,A -85,B 0,C 180,E1 -3512.959,E2 -3512.959} C_VEL
LIN {X 0,Y 544.684,Z 391.057,A -85,B 0,C 180,E1 -3514.07,E2 -3514.07} C_VEL
LIN {X 0,Y 544.653,Z 387.164,A -85,B 0,C 180,E1 -3515.183,E2 -3515.183} C_VEL
LIN {X 0,Y 544.748,Z 381.949,A -85,B 0,C 180,E1 -3516.335,E2 -3516.335} C_VEL
LIN {X 0,Y 544.859,Z 374.595,A -85,B 0,C 180,E1 -3517.598,E2 -3517.598} C_VEL
LIN {X 0,Y 545.016,Z 366.425,A -85,B 0,C 180,E1 -3518.715,E2 -3518.715} C_VEL
LIN {X 0,Y 545.184,Z 358.066,A -85,B 0,C 180,E1 -3519.647,E2 -3519.647} C_VEL
LIN {X 0,Y 545.403,Z 347.752,A -85,B 0,C 180,E1 -3520.581,E2 -3520.581} C_VEL
LIN {X 0,Y 545.596,Z 336.376,A -85,B 0,C 180,E1 -3521.406,E2 -3521.406} C_VEL
LIN {X 0,Y 545.819,Z 324.556,A -85,B 0,C 180,E1 -3522.078,E2 -3522.078} C_VEL
LIN {X 0,Y 546.004,Z 312.541,A -85,B 0,C 180,E1 -3522.592,E2 -3522.592} C_VEL
LIN {X 0,Y 546.151,Z 299.481,A -85,B 0,C 180,E1 -3522.991,E2 -3522.991} C_VEL
LIN {X 0,Y 546.285,Z 287.058,A -85,B 0,C 180,E1 -3523.224,E2 -3523.224} C_VEL
LIN {X 0,Y 546.399,Z 192.693,A -85,B 0,C 180,E1 -3524.473,E2 -3524.473} C_VEL
LIN {X 0,Y 545.3,Z 185.965,A -85,B 0,C 180,E1 -3524.62,E2 -3524.62} C_VEL
LIN {X 0,Y 545.474,Z 170.366,A -85,B 0,C 180,E1 -3527.238,E2 -3527.238} C_VEL
LIN {X 0,Y 545.796,Z 153.999,A -85,B 0,C 180,E1 -3530.06,E2 -3530.06} C_VEL
LIN {X 0,Y 545.719,Z 148.993,A -85,B 0,C 180,E1 -3530.939,E2 -3530.939} C_VEL
LIN {X 0,Y 545.082,Z 145.638,A -85,B 0,C 180,E1 -3531.603,E2 -3531.603} C_VEL
LIN {X 0,Y 545.051,Z 145.594,A -85,B 0,C 180,E1 -3534.369,E2 -3534.369} C_VEL
LIN {X 0,Y 545.086,Z 145.583,A -85,B 0,C 180,E1 -3537.171,E2 -3537.171} C_VEL
LIN {X 0,Y 545.065,Z 145.585,A -85,B 0,C 180,E1 -3539.338,E2 -3539.338} C_VEL
LIN {X 0,Y 545.056,Z 145.587,A -85,B 0,C 180,E1 -3541.914,E2 -3541.914} C_VEL
LIN {X 0,Y 545.076,Z 145.585,A -85,B 0,C 180,E1 -3544.563,E2 -3544.563} C_VEL
LIN {X 0,Y 545.037,Z 145.588,A -85,B 0,C 180,E1 -3547.303,E2 -3547.303} C_VEL
LIN {X 0,Y 545.064,Z 145.587,A -85,B 0,C 180,E1 -3550.142,E2 -3550.142} C_VEL
LIN {X 0,Y 545.077,Z 145.583,A -85,B 0,C 180,E1 -3553.106,E2 -3553.106} C_VEL
LIN {X 0,Y 545.047,Z 145.588,A -85,B 0,C 180,E1 -3556.226,E2 -3556.226} C_VEL
LIN {X 0,Y 545.091,Z 145.58,A -85,B 0,C 180,E1 -3558.886,E2 -3558.886} C_VEL
LIN {X 0,Y 545.048,Z 145.592,A -85,B 0,C 180,E1 -3561.762,E2 -3561.762} C_VEL
LIN {X 0,Y 545.048,Z 145.578,A -85,B 0,C 180,E1 -3564.532,E2 -3564.532} C_VEL
LIN {X 0,Y 545.064,Z 145.582,A -85,B 0,C 180,E1 -3567.211,E2 -3567.211} C_VEL
LIN {X 0,Y 545.058,Z 145.593,A -85,B 0,C 180,E1 -3569.81,E2 -3569.81} C_VEL
LIN {X 0,Y 545.088,Z 145.582,A -85,B 0,C 180,E1 -3572.344,E2 -3572.344} C_VEL
LIN {X 0,Y 545.099,Z 145.58,A -85,B 0,C 180,E1 -3574.819,E2 -3574.819} C_VEL
LIN {X 0,Y 545.03,Z 145.589,A -85,B 0,C 180,E1 -3577.242,E2 -3577.242} C_VEL
LIN {X 0,Y 545.109,Z 145.58,A -85,B 0,C 180,E1 -3580.414,E2 -3580.414} C_VEL
LIN {X 0,Y 545.067,Z 145.589,A -85,B 0,C 180,E1 -3583.521,E2 -3583.521} C_VEL
LIN {X 0,Y 545.087,Z 145.589,A -85,B 0,C 180,E1 -3585.82,E2 -3585.82} C_VEL
LIN {X 0,Y 545.11,Z 145.578,A -85,B 0,C 180,E1 -3588.849,E2 -3588.849} C_VEL
LIN {X 0,Y 545.121,Z 145.582,A -85,B 0,C 180,E1 -3591.847,E2 -3591.847} C_VEL
LIN {X 0,Y 545.195,Z 145.568,A -85,B 0,C 180,E1 -3594.823,E2 -3594.823} C_VEL
LIN {X 0,Y 545.181,Z 145.573,A -85,B 0,C 180,E1 -3597.784,E2 -3597.784} C_VEL
LIN {X 0,Y 545.203,Z 145.567,A -85,B 0,C 180,E1 -3600.739,E2 -3600.739} C_VEL
LIN {X 0,Y 545.163,Z 145.573,A -85,B 0,C 180,E1 -3602.956,E2 -3602.956} C_VEL
LIN {X 0,Y 545.158,Z 145.574,A -85,B 0,C 180,E1 -3605.92,E2 -3605.92} C_VEL
LIN {X 0,Y 545.096,Z 145.583,A -85,B 0,C 180,E1 -3608.9,E2 -3608.9} C_VEL
LIN {X 0,Y 545.098,Z 145.58,A -85,B 0,C 180,E1 -3611.905,E2 -3611.905} C_VEL
LIN {X 0,Y 545.077,Z 145.586,A -85,B 0,C 180,E1 -3614.944,E2 -3614.944} C_VEL
LIN {X 0,Y 545.062,Z 145.582,A -85,B 0,C 180,E1 -3618.026,E2 -3618.026} C_VEL
LIN {X 0,Y 545.084,Z 145.582,A -85,B 0,C 180,E1 -3620.373,E2 -3620.373} C_VEL
LIN {X 0,Y 545.072,Z 145.585,A -85,B 0,C 180,E1 -3623.56,E2 -3623.56} C_VEL
LIN {X 0,Y 545.071,Z 145.584,A -85,B 0,C 180,E1 -3626.001,E2 -3626.001} C_VEL
LIN {X 0,Y 545.068,Z 145.587,A -85,B 0,C 180,E1 -3628.746,E2 -3628.746} C_VEL
LIN {X 0,Y 545.052,Z 145.588,A -85,B 0,C 180,E1 -3631.679,E2 -3631.679} C_VEL
LIN {X 0,Y 545.054,Z 145.586,A -85,B 0,C 180,E1 -3634.565,E2 -3634.565} C_VEL
LIN {X 0,Y 545.03,Z 145.59,A -85,B 0,C 180,E1 -3637.305,E2 -3637.305} C_VEL
LIN {X 0,Y 545.06,Z 145.585,A -85,B 0,C 180,E1 -3640.143,E2 -3640.143} C_VEL
LIN {X 0,Y 545.034,Z 145.593,A -85,B 0,C 180,E1 -3642.695,E2 -3642.695} C_VEL
LIN {X 0,Y 545.026,Z 145.595,A -85,B 0,C 180,E1 -3645.171,E2 -3645.171} C_VEL
LIN {X 0,Y 545.049,Z 145.586,A -85,B 0,C 180,E1 -3647.895,E2 -3647.895} C_VEL
LIN {X 0,Y 545.078,Z 145.587,A -85,B 0,C 180,E1 -3650.819,E2 -3650.819} C_VEL
LIN {X 0,Y 545.032,Z 145.589,A -85,B 0,C 180,E1 -3653.62,E2 -3653.62} C_VEL
LIN {X 0,Y 545.062,Z 145.586,A -85,B 0,C 180,E1 -3656.328,E2 -3656.328} C_VEL
LIN {X 0,Y 545.062,Z 145.59,A -85,B 0,C 180,E1 -3658.952,E2 -3658.952} C_VEL
LIN {X 0,Y 545.08,Z 145.582,A -85,B 0,C 180,E1 -3661.507,E2 -3661.507} C_VEL
LIN {X 0,Y 545.053,Z 145.587,A -85,B 0,C 180,E1 -3663.998,E2 -3663.998} C_VEL
LIN {X 0,Y 545.064,Z 145.627,A -85,B 0,C 180,E1 -3667.294,E2 -3667.294} C_VEL
LIN {X 0,Y 545.416,Z 147.415,A -85,B 0,C 180,E1 -3667.659,E2 -3667.659} C_VEL
LIN {X 0,Y 546.013,Z 152.194,A -85,B 0,C 180,E1 -3668.48,E2 -3668.48} C_VEL
LIN {X 0,Y 545.707,Z 168.904,A -85,B 0,C 180,E1 -3671.218,E2 -3671.218} C_VEL
LIN {X 0,Y 545.397,Z 185.607,A -85,B 0,C 180,E1 -3673.916,E2 -3673.916} C_VEL
LIN {X 0,Y 545.362,Z 195.234,A -85,B 0,C 180,E1 -3675.423,E2 -3675.423} C_VEL
LIN {X 0,Y 546.419,Z 202.349,A -85,B 0,C 180,E1 -3675.573,E2 -3675.573} C_VEL
LIN {X 0,Y 546.255,Z 302.815,A -85,B 0,C 180,E1 -3676.917,E2 -3676.917} C_VEL
LIN {X 0,Y 546.09,Z 316.091,A -85,B 0,C 180,E1 -3677.244,E2 -3677.244} C_VEL
LIN {X 0,Y 545.862,Z 329.37,A -85,B 0,C 180,E1 -3677.735,E2 -3677.735} C_VEL
LIN {X 0,Y 545.706,Z 341.253,A -85,B 0,C 180,E1 -3678.341,E2 -3678.341} C_VEL
LIN {X 0,Y 545.463,Z 353.385,A -85,B 0,C 180,E1 -3679.138,E2 -3679.138} C_VEL
LIN {X 0,Y 545.237,Z 363.559,A -85,B 0,C 180,E1 -3679.979,E2 -3679.979} C_VEL
LIN {X 0,Y 545.054,Z 372.711,A -85,B 0,C 180,E1 -3680.912,E2 -3680.912} C_VEL
LIN {X 0,Y 544.916,Z 381.626,A -85,B 0,C 180,E1 -3682.03,E2 -3682.03} C_VEL
LIN {X 0,Y 544.767,Z 388.798,A -85,B 0,C 180,E1 -3683.146,E2 -3683.146} C_VEL
LIN {X 0,Y 544.741,Z 395.328,A -85,B 0,C 180,E1 -3684.447,E2 -3684.447} C_VEL
LIN {X 0,Y 544.659,Z 399.647,A -85,B 0,C 180,E1 -3685.559,E2 -3685.559} C_VEL
LIN {X 0,Y 544.669,Z 401.932,A -85,B 0,C 180,E1 -3686.301,E2 -3686.301} C_VEL
LIN {X 0,Y 544.65,Z 403.785,A -85,B 0,C 180,E1 -3687.041,E2 -3687.041} C_VEL
LIN {X 0,Y 544.546,Z 406.164,A -85,B 0,C 180,E1 -3688.521,E2 -3688.521} C_VEL
LIN {X 0,Y 544.541,Z 406.985,A -85,B 0,C 180,E1 -3690,E2 -3690} C_VEL
LIN {X 0,Y 544.546,Z 406.166,A -85,B 0,C 180,E1 -3691.479,E2 -3691.479} C_VEL
LIN {X 0,Y 544.65,Z 403.79,A -85,B 0,C 180,E1 -3692.958,E2 -3692.958} C_VEL
LIN {X 0,Y 544.684,Z 400.87,A -85,B 0,C 180,E1 -3694.069,E2 -3694.069} C_VEL
LIN {X 0,Y 544.653,Z 396.915,A -85,B 0,C 180,E1 -3695.182,E2 -3695.182} C_VEL
LIN {X 0,Y 544.733,Z 391.558,A -85,B 0,C 180,E1 -3696.347,E2 -3696.347} C_VEL
LIN {X 0,Y 544.859,Z 384.182,A -85,B 0,C 180,E1 -3697.597,E2 -3697.597} C_VEL
LIN {X 0,Y 545.012,Z 375.927,A -85,B 0,C 180,E1 -3698.714,E2 -3698.714} C_VEL
LIN {X 0,Y 545.18,Z 367.465,A -85,B 0,C 180,E1 -3699.647,E2 -3699.647} C_VEL
LIN {X 0,Y 545.395,Z 357.005,A -85,B 0,C 180,E1 -3700.58,E2 -3700.58} C_VEL
LIN {X 0,Y 545.621,Z 345.255,A -85,B 0,C 180,E1 -3701.42,E2 -3701.42} C_VEL
LIN {X 0,Y 545.848,Z 333.384,A -85,B 0,C 180,E1 -3702.076,E2 -3702.076} C_VEL
LIN {X 0,Y 546.029,Z 321.058,A -85,B 0,C 180,E1 -3702.591,E2 -3702.591} C_VEL
LIN {X 0,Y 546.198,Z 308.411,A -85,B 0,C 180,E1 -3702.965,E2 -3702.965} C_VEL
LIN {X 0,Y 546.298,Z 295.226,A -85,B 0,C 180,E1 -3703.199,E2 -3703.199} C_VEL
LIN {X 0,Y 546.419,Z 202.398,A -85,B 0,C 180,E1 -3704.427,E2 -3704.427} C_VEL
LIN {X 0,Y 545.361,Z 195.255,A -85,B 0,C 180,E1 -3704.577,E2 -3704.577} C_VEL
LIN {X 0,Y 545.68,Z 173.681,A -85,B 0,C 180,E1 -3708.004,E2 -3708.004} C_VEL
LIN {X 0,Y 545.967,Z 154.586,A -85,B 0,C 180,E1 -3711.126,E2 -3711.126} C_VEL
LIN {X 0,Y 545.777,Z 149.338,A -85,B 0,C 180,E1 -3712.005,E2 -3712.005} C_VEL
LIN {X 0,Y 545.096,Z 145.759,A -85,B 0,C 180,E1 -3712.654,E2 -3712.654} C_VEL
LIN {X 0,Y 545.036,Z 145.595,A -85,B 0,C 180,E1 -3715.495,E2 -3715.495} C_VEL
LIN {X 0,Y 545.054,Z 145.59,A -85,B 0,C 180,E1 -3717.657,E2 -3717.657} C_VEL
LIN {X 0,Y 545.042,Z 145.587,A -85,B 0,C 180,E1 -3720.239,E2 -3720.239} C_VEL
LIN {X 0,Y 545.073,Z 145.591,A -85,B 0,C 180,E1 -3723.061,E2 -3723.061} C_VEL
LIN {X 0,Y 545.02,Z 145.593,A -85,B 0,C 180,E1 -3725.671,E2 -3725.671} C_VEL
LIN {X 0,Y 545.044,Z 145.582,A -85,B 0,C 180,E1 -3728.237,E2 -3728.237} C_VEL
LIN {X 0,Y 545.074,Z 145.584,A -85,B 0,C 180,E1 -3730.472,E2 -3730.472} C_VEL
LIN {X 0,Y 545.038,Z 145.595,A -85,B 0,C 180,E1 -3733.109,E2 -3733.109} C_VEL
LIN {X 0,Y 545.042,Z 145.587,A -85,B 0,C 180,E1 -3735.869,E2 -3735.869} C_VEL
LIN {X 0,Y 545.072,Z 145.59,A -85,B 0,C 180,E1 -3738.884,E2 -3738.884} C_VEL
LIN {X 0,Y 545.07,Z 145.59,A -85,B 0,C 180,E1 -3740.817,E2 -3740.817} C_VEL
LIN {X 0,Y 545.033,Z 145.582,A -85,B 0,C 180,E1 -3743.619,E2 -3743.619} C_VEL
LIN {X 0,Y 545.041,Z 145.587,A -85,B 0,C 180,E1 -3746.326,E2 -3746.326} C_VEL
LIN {X 0,Y 545.053,Z 145.593,A -85,B 0,C 180,E1 -3748.951,E2 -3748.951} C_VEL
LIN {X 0,Y 545.072,Z 145.584,A -85,B 0,C 180,E1 -3751.506,E2 -3751.506} C_VEL
LIN {X 0,Y 545.074,Z 145.587,A -85,B 0,C 180,E1 -3754.493,E2 -3754.493} C_VEL
LIN {X 0,Y 545.024,Z 145.592,A -85,B 0,C 180,E1 -3757.242,E2 -3757.242} C_VEL
LIN {X 0,Y 545.107,Z 145.583,A -85,B 0,C 180,E1 -3760.414,E2 -3760.414} C_VEL
LIN {X 0,Y 545.058,Z 145.585,A -85,B 0,C 180,E1 -3763.521,E2 -3763.521} C_VEL
LIN {X 0,Y 545.08,Z 145.582,A -85,B 0,C 180,E1 -3765.819,E2 -3765.819} C_VEL
LIN {X 0,Y 545.135,Z 145.58,A -85,B 0,C 180,E1 -3768.85,E2 -3768.85} C_VEL
LIN {X 0,Y 545.108,Z 145.579,A -85,B 0,C 180,E1 -3771.847,E2 -3771.847} C_VEL
LIN {X 0,Y 545.19,Z 145.57,A -85,B 0,C 180,E1 -3774.823,E2 -3774.823} C_VEL
LIN {X 0,Y 545.174,Z 145.57,A -85,B 0,C 180,E1 -3777.784,E2 -3777.784} C_VEL
LIN {X 0,Y 545.205,Z 145.57,A -85,B 0,C 180,E1 -3780.739,E2 -3780.739} C_VEL
LIN {X 0,Y 545.162,Z 145.572,A -85,B 0,C 180,E1 -3782.956,E2 -3782.956} C_VEL
LIN {X 0,Y 545.152,Z 145.575,A -85,B 0,C 180,E1 -3785.92,E2 -3785.92} C_VEL
LIN {X 0,Y 545.107,Z 145.577,A -85,B 0,C 180,E1 -3788.9,E2 -3788.9} C_VEL
LIN {X 0,Y 545.122,Z 145.579,A -85,B 0,C 180,E1 -3791.905,E2 -3791.905} C_VEL
LIN {X 0,Y 545.073,Z 145.581,A -85,B 0,C 180,E1 -3794.944,E2 -3794.944} C_VEL
LIN {X 0,Y 545.066,Z 145.588,A -85,B 0,C 180,E1 -3798.026,E2 -3798.026} C_VEL
LIN {X 0,Y 545.087,Z 145.587,A -85,B 0,C 180,E1 -3800.373,E2 -3800.373} C_VEL
LIN {X 0,Y 545.082,Z 145.582,A -85,B 0,C 180,E1 -3803.559,E2 -3803.559} C_VEL
LIN {X 0,Y 545.067,Z 145.591,A -85,B 0,C 180,E1 -3806.001,E2 -3806.001} C_VEL
LIN {X 0,Y 545.08,Z 145.583,A -85,B 0,C 180,E1 -3808.749,E2 -3808.749} C_VEL
LIN {X 0,Y 545.047,Z 145.589,A -85,B 0,C 180,E1 -3811.68,E2 -3811.68} C_VEL
LIN {X 0,Y 545.067,Z 145.577,A -85,B 0,C 180,E1 -3814.564,E2 -3814.564} C_VEL
LIN {X 0,Y 545.053,Z 145.582,A -85,B 0,C 180,E1 -3817.027,E2 -3817.027} C_VEL
LIN {X 0,Y 544.346,Z 145.675,A -85,B 0,C 180,E1 -3817.644,E2 -3817.644} C_VEL
LIN {X 0,Y 541.482,Z 146.032,A -85,B 0,C 180,E1 -3818.645,E2 -3818.645} C_VEL
LIN {X 0,Y 539.096,Z 146.331,A -85,B 0,C 180,E1 -3819.45,E2 -3819.45} C_VEL
LIN {X 0,Y 538.088,Z 146.461,A -85,B 0,C 180,E1 -3820.072,E2 -3820.072} C_VEL
LIN {X 0,Y 538.013,Z 146.463,A -85,B 0,C 180,E1 -3820.283,E2 -3820.283} C_VEL
LIN {X 0,Y 538.019,Z 146.456,A -85,B 0,C 180,E1 -3822.989,E2 -3822.989} C_VEL
LIN {X 0,Y 537.997,Z 146.47,A -85,B 0,C 180,E1 -3826.185,E2 -3826.185} C_VEL
LIN {X 0,Y 538.043,Z 146.458,A -85,B 0,C 180,E1 -3829.254,E2 -3829.254} C_VEL
LIN {X 0,Y 537.987,Z 146.472,A -85,B 0,C 180,E1 -3832.123,E2 -3832.123} C_VEL
LIN {X 0,Y 538.004,Z 146.461,A -85,B 0,C 180,E1 -3834.917,E2 -3834.917} C_VEL
LIN {X 0,Y 538.016,Z 146.47,A -85,B 0,C 180,E1 -3837.618,E2 -3837.618} C_VEL
LIN {X 0,Y 538.014,Z 146.466,A -85,B 0,C 180,E1 -3840.24,E2 -3840.24} C_VEL
LIN {X 0,Y 538.049,Z 146.46,A -85,B 0,C 180,E1 -3842.796,E2 -3842.796} C_VEL
LIN {X 0,Y 538.047,Z 146.464,A -85,B 0,C 180,E1 -3845.294,E2 -3845.294} C_VEL
LIN {X 0,Y 538.076,Z 146.662,A -85,B 0,C 180,E1 -3848.405,E2 -3848.405} C_VEL
LIN {X 0,Y 538.896,Z 151.866,A -85,B 0,C 180,E1 -3849.384,E2 -3849.384} C_VEL
LIN {X 0,Y 538.539,Z 168.521,A -85,B 0,C 180,E1 -3852.3,E2 -3852.3} C_VEL
LIN {X 0,Y 538.272,Z 185.808,A -85,B 0,C 180,E1 -3855.256,E2 -3855.256} C_VEL
LIN {X 0,Y 538.682,Z 188.518,A -85,B 0,C 180,E1 -3855.349,E2 -3855.349} C_VEL
LIN {X 0,Y 539.628,Z 194.544,A -85,B 0,C 180,E1 -3855.456,E2 -3855.456} C_VEL
LIN {X 0,Y 539.402,Z 293.316,A -85,B 0,C 180,E1 -3856.797,E2 -3856.797} C_VEL
LIN {X 0,Y 539.199,Z 305.754,A -85,B 0,C 180,E1 -3857.103,E2 -3857.103} C_VEL
LIN {X 0,Y 538.963,Z 318.632,A -85,B 0,C 180,E1 -3857.576,E2 -3857.576} C_VEL
LIN {X 0,Y 538.815,Z 329.825,A -85,B 0,C 180,E1 -3858.133,E2 -3858.133} C_VEL
LIN {X 0,Y 538.577,Z 340.473,A -85,B 0,C 180,E1 -3858.808,E2 -3858.808} C_VEL
LIN {X 0,Y 538.31,Z 351.196,A -85,B 0,C 180,E1 -3859.659,E2 -3859.659} C_VEL
LIN {X 0,Y 538.085,Z 360.845,A -85,B 0,C 180,E1 -3860.604,E2 -3860.604} C_VEL
LIN {X 0,Y 537.937,Z 368.751,A -85,B 0,C 180,E1 -3861.549,E2 -3861.549} C_VEL
LIN {X 0,Y 537.759,Z 376.485,A -85,B 0,C 180,E1 -3862.68,E2 -3862.68} C_VEL
LIN {X 0,Y 537.729,Z 383.578,A -85,B 0,C 180,E1 -3863.999,E2 -3863.999} C_VEL
LIN {X 0,Y 537.541,Z 388.309,A -85,B 0,C 180,E1 -3865.125,E2 -3865.125} C_VEL
LIN {X 0,Y 537.591,Z 391.932,A -85,B 0,C 180,E1 -3866.253,E2 -3866.253} C_VEL
LIN {X 0,Y 537.58,Z 393.805,A -85,B 0,C 180,E1 -3867.003,E2 -3867.003} C_VEL
LIN {X 0,Y 537.49,Z 395.221,A -85,B 0,C 180,E1 -3867.752,E2 -3867.752} C_VEL
LIN {X 0,Y 537.443,Z 396.846,A -85,B 0,C 180,E1 -3869.251,E2 -3869.251} C_VEL
LIN {X 0,Y 537.443,Z 397.085,A -85,B 0,C 180,E1 -3870,E2 -3870} C_VEL
LIN {X 0,Y 537.442,Z 396.903,A -85,B 0,C 180,E1 -3870.75,E2 -3870.75} C_VEL
LIN {X 0,Y 537.49,Z 395.351,A -85,B 0,C 180,E1 -3872.248,E2 -3872.248} C_VEL
LIN {X 0,Y 537.58,Z 393.992,A -85,B 0,C 180,E1 -3872.998,E2 -3872.998} C_VEL
LIN {X 0,Y 537.604,Z 391.121,A -85,B 0,C 180,E1 -3874.123,E2 -3874.123} C_VEL
LIN {X 0,Y 537.587,Z 387.227,A -85,B 0,C 180,E1 -3875.251,E2 -3875.251} C_VEL
LIN {X 0,Y 537.661,Z 382.382,A -85,B 0,C 180,E1 -3876.342,E2 -3876.342} C_VEL
LIN {X 0,Y 537.79,Z 375.882,A -85,B 0,C 180,E1 -3877.509,E2 -3877.509} C_VEL
LIN {X 0,Y 537.961,Z 367.968,A -85,B 0,C 180,E1 -3878.641,E2 -3878.641} C_VEL
LIN {X 0,Y 538.153,Z 358.125,A -85,B 0,C 180,E1 -3879.775,E2 -3879.775} C_VEL
LIN {X 0,Y 538.396,Z 347.81,A -85,B 0,C 180,E1 -3880.72,E2 -3880.72} C_VEL
LIN {X 0,Y 538.62,Z 336.805,A -85,B 0,C 180,E1 -3881.53,E2 -3881.53} C_VEL
LIN {X 0,Y 538.869,Z 326.421,A -85,B 0,C 180,E1 -3882.14,E2 -3882.14} C_VEL
LIN {X 0,Y 539.032,Z 315.105,A -85,B 0,C 180,E1 -3882.662,E2 -3882.662} C_VEL
LIN {X 0,Y 539.214,Z 302.269,A -85,B 0,C 180,E1 -3883.089,E2 -3883.089} C_VEL
LIN {X 0,Y 539.362,Z 288.617,A -85,B 0,C 180,E1 -3883.373,E2 -3883.373} C_VEL
LIN {X 0,Y 539.493,Z 193.151,A -85,B 0,C 180,E1 -3884.656,E2 -3884.656} C_VEL
LIN {X 0,Y 538.312,Z 186.326,A -85,B 0,C 180,E1 -3884.798,E2 -3884.798} C_VEL
LIN {X 0,Y 538.246,Z 185.129,A -85,B 0,C 180,E1 -3884.931,E2 -3884.931} C_VEL
LIN {X 0,Y 538.512,Z 169.094,A -85,B 0,C 180,E1 -3887.691,E2 -3887.691} C_VEL
LIN {X 0,Y 538.895,Z 151.242,A -85,B 0,C 180,E1 -3890.817,E2 -3890.817} C_VEL
LIN {X 0,Y 538.033,Z 146.518,A -85,B 0,C 180,E1 -3891.742,E2 -3891.742} C_VEL
LIN {X 0,Y 538.05,Z 146.465,A -85,B 0,C 180,E1 -3894.707,E2 -3894.707} C_VEL
LIN {X 0,Y 538.051,Z 146.46,A -85,B 0,C 180,E1 -3897.35,E2 -3897.35} C_VEL
LIN {X 0,Y 538.017,Z 146.465,A -85,B 0,C 180,E1 -3899.761,E2 -3899.761} C_VEL
LIN {X 0,Y 538.019,Z 146.471,A -85,B 0,C 180,E1 -3902.382,E2 -3902.382} C_VEL
LIN {X 0,Y 538.012,Z 146.46,A -85,B 0,C 180,E1 -3905.083,E2 -3905.083} C_VEL
LIN {X 0,Y 537.991,Z 146.47,A -85,B 0,C 180,E1 -3907.877,E2 -3907.877} C_VEL
LIN {X 0,Y 538.047,Z 146.457,A -85,B 0,C 180,E1 -3910.775,E2 -3910.775} C_VEL
LIN {X 0,Y 538.019,Z 146.471,A -85,B 0,C 180,E1 -3914.073,E2 -3914.073} C_VEL
LIN {X 0,Y 538.009,Z 146.457,A -85,B 0,C 180,E1 -3917.213,E2 -3917.213} C_VEL
LIN {X 0,Y 538.023,Z 146.469,A -85,B 0,C 180,E1 -3920.203,E2 -3920.203} C_VEL
LIN {X 0,Y 538.023,Z 146.458,A -85,B 0,C 180,E1 -3923.067,E2 -3923.067} C_VEL
LIN {X 0,Y 538.016,Z 146.458,A -85,B 0,C 180,E1 -3925.826,E2 -3925.826} C_VEL
LIN {X 0,Y 538.003,Z 146.466,A -85,B 0,C 180,E1 -3928.498,E2 -3928.498} C_VEL
LIN {X 0,Y 538.055,Z 146.457,A -85,B 0,C 180,E1 -3931.099,E2 -3931.099} C_VEL
LIN {X 0,Y 538.035,Z 146.463,A -85,B 0,C 180,E1 -3933.633,E2 -3933.633} C_VEL
LIN {X 0,Y 538,Z 146.468,A -85,B 0,C 180,E1 -3936.122,E2 -3936.122} C_VEL
LIN {X 0,Y 538.031,Z 146.461,A -85,B 0,C 180,E1 -3939.348,E2 -3939.348} C_VEL
LIN {X 0,Y 538.047,Z 146.458,A -85,B 0,C 180,E1 -3942.517,E2 -3942.517} C_VEL
LIN {X 0,Y 538.056,Z 146.462,A -85,B 0,C 180,E1 -3945.63,E2 -3945.63} C_VEL
LIN {X 0,Y 538.069,Z 146.455,A -85,B 0,C 180,E1 -3948.701,E2 -3948.701} C_VEL
LIN {X 0,Y 538.078,Z 146.461,A -85,B 0,C 180,E1 -3951.739,E2 -3951.739} C_VEL
LIN {X 0,Y 538.152,Z 146.445,A -85,B 0,C 180,E1 -3954.755,E2 -3954.755} C_VEL
LIN {X 0,Y 538.154,Z 146.449,A -85,B 0,C 180,E1 -3957.755,E2 -3957.755} C_VEL
LIN {X 0,Y 538.174,Z 146.443,A -85,B 0,C 180,E1 -3960.748,E2 -3960.748} C_VEL
LIN {X 0,Y 538.129,Z 146.45,A -85,B 0,C 180,E1 -3962.994,E2 -3962.994} C_VEL
LIN {X 0,Y 538.109,Z 146.452,A -85,B 0,C 180,E1 -3965.997,E2 -3965.997} C_VEL
LIN {X 0,Y 538.05,Z 146.462,A -85,B 0,C 180,E1 -3969.018,E2 -3969.018} C_VEL
LIN {X 0,Y 538.058,Z 146.456,A -85,B 0,C 180,E1 -3972.063,E2 -3972.063} C_VEL
LIN {X 0,Y 538.037,Z 146.466,A -85,B 0,C 180,E1 -3975.144,E2 -3975.144} C_VEL
LIN {X 0,Y 538.017,Z 146.459,A -85,B 0,C 180,E1 -3978.271,E2 -3978.271} C_VEL
LIN {X 0,Y 538.029,Z 146.462,A -85,B 0,C 180,E1 -3980.652,E2 -3980.652} C_VEL
LIN {X 0,Y 537.995,Z 146.463,A -85,B 0,C 180,E1 -3983.889,E2 -3983.889} C_VEL
LIN {X 0,Y 538.033,Z 146.46,A -85,B 0,C 180,E1 -3986.367,E2 -3986.367} C_VEL
LIN {X 0,Y 538.024,Z 146.467,A -85,B 0,C 180,E1 -3988.934,E2 -3988.934} C_VEL
LIN {X 0,Y 538.003,Z 146.465,A -85,B 0,C 180,E1 -3991.887,E2 -3991.887} C_VEL
LIN {X 0,Y 538.004,Z 146.465,A -85,B 0,C 180,E1 -3994.618,E2 -3994.618} C_VEL
LIN {X 0,Y 537.999,Z 146.465,A -85,B 0,C 180,E1 -3997.17,E2 -3997.17} C_VEL
LIN {X 0,Y 538.016,Z 146.462,A -85,B 0,C 180,E1 -3999.798,E2 -3999.798} C_VEL
LIN {X 0,Y 537.984,Z 146.473,A -85,B 0,C 180,E1 -4002.79,E2 -4002.79} C_VEL
LIN {X 0,Y 537.997,Z 146.471,A -85,B 0,C 180,E1 -4005.138,E2 -4005.138} C_VEL
LIN {X 0,Y 537.997,Z 146.466,A -85,B 0,C 180,E1 -4008.224,E2 -4008.224} C_VEL
LIN {X 0,Y 538.01,Z 146.463,A -85,B 0,C 180,E1 -4011.17,E2 -4011.17} C_VEL
LIN {X 0,Y 537.988,Z 146.467,A -85,B 0,C 180,E1 -4014.09,E2 -4014.09} C_VEL
LIN {X 0,Y 538.03,Z 146.466,A -85,B 0,C 180,E1 -4016.728,E2 -4016.728} C_VEL
LIN {X 0,Y 538.006,Z 146.464,A -85,B 0,C 180,E1 -4019.561,E2 -4019.561} C_VEL
LIN {X 0,Y 538.019,Z 146.462,A -85,B 0,C 180,E1 -4021.949,E2 -4021.949} C_VEL
LIN {X 0,Y 538.02,Z 146.468,A -85,B 0,C 180,E1 -4024.465,E2 -4024.465} C_VEL
LIN {X 0,Y 538.021,Z 146.617,A -85,B 0,C 180,E1 -4027.183,E2 -4027.183} C_VEL
LIN {X 0,Y 539.068,Z 152.249,A -85,B 0,C 180,E1 -4028.208,E2 -4028.208} C_VEL
LIN {X 0,Y 538.746,Z 167.649,A -85,B 0,C 180,E1 -4030.768,E2 -4030.768} C_VEL
LIN {X 0,Y 538.476,Z 181.965,A -85,B 0,C 180,E1 -4033.118,E2 -4033.118} C_VEL
LIN {X 0,Y 538.32,Z 195.214,A -85,B 0,C 180,E1 -4035.231,E2 -4035.231} C_VEL
LIN {X 0,Y 539.676,Z 204.119,A -85,B 0,C 180,E1 -4035.413,E2 -4035.413} C_VEL
LIN {X 0,Y 539.349,Z 302.75,A -85,B 0,C 180,E1 -4036.747,E2 -4036.747} C_VEL
LIN {X 0,Y 539.164,Z 316.026,A -85,B 0,C 180,E1 -4037.078,E2 -4037.078} C_VEL
LIN {X 0,Y 538.906,Z 329.305,A -85,B 0,C 180,E1 -4037.574,E2 -4037.574} C_VEL
LIN {X 0,Y 538.719,Z 341.188,A -85,B 0,C 180,E1 -4038.188,E2 -4038.188} C_VEL
LIN {X 0,Y 538.486,Z 353.32,A -85,B 0,C 180,E1 -4038.996,E2 -4038.996} C_VEL
LIN {X 0,Y 538.231,Z 363.494,A -85,B 0,C 180,E1 -4039.847,E2 -4039.847} C_VEL
LIN {X 0,Y 538.019,Z 372.646,A -85,B 0,C 180,E1 -4040.792,E2 -4040.792} C_VEL
LIN {X 0,Y 537.851,Z 381.561,A -85,B 0,C 180,E1 -4041.925,E2 -4041.925} C_VEL
LIN {X 0,Y 537.702,Z 388.733,A -85,B 0,C 180,E1 -4043.056,E2 -4043.056} C_VEL
LIN {X 0,Y 537.676,Z 395.263,A -85,B 0,C 180,E1 -4044.374,E2 -4044.374} C_VEL
LIN {X 0,Y 537.555,Z 399.581,A -85,B 0,C 180,E1 -4045.501,E2 -4045.501} C_VEL
LIN {X 0,Y 537.591,Z 401.867,A -85,B 0,C 180,E1 -4046.252,E2 -4046.252} C_VEL
LIN {X 0,Y 537.551,Z 403.72,A -85,B 0,C 180,E1 -4047.002,E2 -4047.002} C_VEL
LIN {X 0,Y 537.451,Z 406.099,A -85,B 0,C 180,E1 -4048.501,E2 -4048.501} C_VEL
LIN {X 0,Y 537.442,Z 406.92,A -85,B 0,C 180,E1 -4050,E2 -4050} C_VEL
LIN {X 0,Y 537.451,Z 406.101,A -85,B 0,C 180,E1 -4051.498,E2 -4051.498} C_VEL
LIN {X 0,Y 537.551,Z 403.725,A -85,B 0,C 180,E1 -4052.997,E2 -4052.997} C_VEL
LIN {X 0,Y 537.603,Z 400.805,A -85,B 0,C 180,E1 -4054.123,E2 -4054.123} C_VEL
LIN {X 0,Y 537.587,Z 396.85,A -85,B 0,C 180,E1 -4055.25,E2 -4055.25} C_VEL
LIN {X 0,Y 537.645,Z 391.997,A -85,B 0,C 180,E1 -4056.33,E2 -4056.33} C_VEL
LIN {X 0,Y 537.771,Z 385.35,A -85,B 0,C 180,E1 -4057.509,E2 -4057.509} C_VEL
LIN {X 0,Y 537.963,Z 377.349,A -85,B 0,C 180,E1 -4058.64,E2 -4058.64} C_VEL
LIN {X 0,Y 538.132,Z 369.195,A -85,B 0,C 180,E1 -4059.585,E2 -4059.585} C_VEL
LIN {X 0,Y 538.355,Z 359.247,A -85,B 0,C 180,E1 -4060.53,E2 -4060.53} C_VEL
LIN {X 0,Y 538.573,Z 349.435,A -85,B 0,C 180,E1 -4061.287,E2 -4061.287} C_VEL
LIN {X 0,Y 538.757,Z 338.99,A -85,B 0,C 180,E1 -4061.939,E2 -4061.939} C_VEL
LIN {X 0,Y 538.956,Z 325.93,A -85,B 0,C 180,E1 -4062.568,E2 -4062.568} C_VEL
LIN {X 0,Y 539.236,Z 312.919,A -85,B 0,C 180,E1 -4063.016,E2 -4063.016} C_VEL
LIN {X 0,Y 539.357,Z 299.948,A -85,B 0,C 180,E1 -4063.3,E2 -4063.3} C_VEL
LIN {X 0,Y 539.531,Z 202.87,A -85,B 0,C 180,E1 -4064.608,E2 -4064.608} C_VEL
LIN {X 0,Y 538.338,Z 195.306,A -85,B 0,C 180,E1 -4064.763,E2 -4064.763} C_VEL
LIN {X 0,Y 538.307,Z 191.511,A -85,B 0,C 180,E1 -4065.329,E2 -4065.329} C_VEL
LIN {X 0,Y 538.686,Z 172.425,A -85,B 0,C 180,E1 -4068.443,E2 -4068.443} C_VEL
LIN {X 0,Y 539.016,Z 154.526,A -85,B 0,C 180,E1 -4071.412,E2 -4071.412} C_VEL
LIN {X 0,Y 538.876,Z 150.918,A -85,B 0,C 180,E1 -4072.025,E2 -4072.025} C_VEL
LIN {X 0,Y 538.015,Z 146.557,A -85,B 0,C 180,E1 -4072.842,E2 -4072.842} C_VEL
LIN {X 0,Y 537.996,Z 146.469,A -85,B 0,C 180,E1 -4075.661,E2 -4075.661} C_VEL
LIN {X 0,Y 538.017,Z 146.463,A -85,B 0,C 180,E1 -4078.05,E2 -4078.05} C_VEL
LIN {X 0,Y 538.004,Z 146.464,A -85,B 0,C 180,E1 -4080.627,E2 -4080.627} C_VEL
LIN {X 0,Y 538.042,Z 146.464,A -85,B 0,C 180,E1 -4083.282,E2 -4083.282} C_VEL
LIN {X 0,Y 537.985,Z 146.467,A -85,B 0,C 180,E1 -4086.004,E2 -4086.004} C_VEL
LIN {X 0,Y 538.007,Z 146.463,A -85,B 0,C 180,E1 -4088.829,E2 -4088.829} C_VEL
LIN {X 0,Y 538.007,Z 146.464,A -85,B 0,C 180,E1 -4091.876,E2 -4091.876} C_VEL
LIN {X 0,Y 538.021,Z 146.47,A -85,B 0,C 180,E1 -4095.139,E2 -4095.139} C_VEL
LIN {X 0,Y 538.022,Z 146.461,A -85,B 0,C 180,E1 -4098.226,E2 -4098.226} C_VEL
LIN {X 0,Y 538.003,Z 146.466,A -85,B 0,C 180,E1 -4101.169,E2 -4101.169} C_VEL
LIN {X 0,Y 537.986,Z 146.458,A -85,B 0,C 180,E1 -4104.087,E2 -4104.087} C_VEL
LIN {X 0,Y 538.02,Z 146.466,A -85,B 0,C 180,E1 -4106.727,E2 -4106.727} C_VEL
LIN {X 0,Y 538.002,Z 146.463,A -85,B 0,C 180,E1 -4109.558,E2 -4109.558} C_VEL
LIN {X 0,Y 538.038,Z 146.465,A -85,B 0,C 180,E1 -4112.649,E2 -4112.649} C_VEL
LIN {X 0,Y 538.01,Z 146.463,A -85,B 0,C 180,E1 -4115.291,E2 -4115.291} C_VEL
LIN {X 0,Y 538.002,Z 146.464,A -85,B 0,C 180,E1 -4118.041,E2 -4118.041} C_VEL
LIN {X 0,Y 538.023,Z 146.465,A -85,B 0,C 180,E1 -4120.939,E2 -4120.939} C_VEL
LIN {X 0,Y 538.005,Z 146.464,A -85,B 0,C 180,E1 -4123.298,E2 -4123.298} C_VEL
LIN {X 0,Y 538.049,Z 146.458,A -85,B 0,C 180,E1 -4125.63,E2 -4125.63} C_VEL
LIN {X 0,Y 538.088,Z 146.458,A -85,B 0,C 180,E1 -4128.702,E2 -4128.702} C_VEL
LIN {X 0,Y 538.065,Z 146.456,A -85,B 0,C 180,E1 -4131.739,E2 -4131.739} C_VEL
LIN {X 0,Y 538.147,Z 146.448,A -85,B 0,C 180,E1 -4134.755,E2 -4134.755} C_VEL
LIN {X 0,Y 538.147,Z 146.446,A -85,B 0,C 180,E1 -4137.755,E2 -4137.755} C_VEL
LIN {X 0,Y 538.174,Z 146.445,A -85,B 0,C 180,E1 -4140.748,E2 -4140.748} C_VEL
LIN {X 0,Y 538.127,Z 146.448,A -85,B 0,C 180,E1 -4142.995,E2 -4142.995} C_VEL
LIN {X 0,Y 538.103,Z 146.454,A -85,B 0,C 180,E1 -4145.998,E2 -4145.998} C_VEL
LIN {X 0,Y 538.057,Z 146.454,A -85,B 0,C 180,E1 -4149.018,E2 -4149.018} C_VEL
LIN {X 0,Y 538.07,Z 146.459,A -85,B 0,C 180,E1 -4152.063,E2 -4152.063} C_VEL
LIN {X 0,Y 538.033,Z 146.457,A -85,B 0,C 180,E1 -4155.144,E2 -4155.144} C_VEL
LIN {X 0,Y 538.019,Z 146.47,A -85,B 0,C 180,E1 -4158.271,E2 -4158.271} C_VEL
LIN {X 0,Y 538.031,Z 146.462,A -85,B 0,C 180,E1 -4160.652,E2 -4160.652} C_VEL
LIN {X 0,Y 538.013,Z 146.466,A -85,B 0,C 180,E1 -4163.888,E2 -4163.888} C_VEL
LIN {X 0,Y 538.03,Z 146.465,A -85,B 0,C 180,E1 -4166.367,E2 -4166.367} C_VEL
LIN {X 0,Y 538.022,Z 146.461,A -85,B 0,C 180,E1 -4168.935,E2 -4168.935} C_VEL
LIN {X 0,Y 538,Z 146.47,A -85,B 0,C 180,E1 -4171.888,E2 -4171.888} C_VEL
LIN {X 0,Y 538.017,Z 146.454,A -85,B 0,C 180,E1 -4174.621,E2 -4174.621} C_VEL
LIN {X 0,Y 537.997,Z 146.461,A -85,B 0,C 180,E1 -4177.171,E2 -4177.171} C_VEL
LIN {X 0,Y 538.013,Z 146.463,A -85,B 0,C 180,E1 -4180.283,E2 -4180.283} C_VEL
LIN {X 0,Y 537.364,Z 146.544,A -85,B 0,C 180,E1 -4180.908,E2 -4180.908} C_VEL
LIN {X 0,Y 534.509,Z 146.904,A -85,B 0,C 180,E1 -4181.923,E2 -4181.923} C_VEL
LIN {X 0,Y 532.081,Z 147.202,A -85,B 0,C 180,E1 -4182.74,E2 -4182.74} C_VEL
LIN {X 0,Y 531.032,Z 147.329,A -85,B 0,C 180,E1 -4183.371,E2 -4183.371} C_VEL
LIN {X 0,Y 530.944,Z 147.339,A -85,B 0,C 180,E1 -4183.585,E2 -4183.585} C_VEL
LIN {X 0,Y 530.948,Z 147.345,A -85,B 0,C 180,E1 -4186.505,E2 -4186.505} C_VEL
LIN {X 0,Y 530.98,Z 147.336,A -85,B 0,C 180,E1 -4188.977,E2 -4188.977} C_VEL
LIN {X 0,Y 530.951,Z 147.343,A -85,B 0,C 180,E1 -4191.53,E2 -4191.53} C_VEL
LIN {X 0,Y 530.971,Z 147.339,A -85,B 0,C 180,E1 -4194.383,E2 -4194.383} C_VEL
LIN {X 0,Y 530.964,Z 147.343,A -85,B 0,C 180,E1 -4197.134,E2 -4197.134} C_VEL
LIN {X 0,Y 530.968,Z 147.348,A -85,B 0,C 180,E1 -4199.804,E2 -4199.804} C_VEL
LIN {X 0,Y 531.009,Z 147.338,A -85,B 0,C 180,E1 -4202.469,E2 -4202.469} C_VEL
LIN {X 0,Y 531.004,Z 147.339,A -85,B 0,C 180,E1 -4204.943,E2 -4204.943} C_VEL
LIN {X 0,Y 531.038,Z 147.498,A -85,B 0,C 180,E1 -4208.25,E2 -4208.25} C_VEL
LIN {X 0,Y 531.939,Z 152.942,A -85,B 0,C 180,E1 -4209.294,E2 -4209.294} C_VEL
LIN {X 0,Y 531.523,Z 171.002,A -85,B 0,C 180,E1 -4212.495,E2 -4212.495} C_VEL
LIN {X 0,Y 531.265,Z 185.967,A -85,B 0,C 180,E1 -4215.067,E2 -4215.067} C_VEL
LIN {X 0,Y 532.04,Z 190.584,A -85,B 0,C 180,E1 -4215.188,E2 -4215.188} C_VEL
LIN {X 0,Y 532.763,Z 195.397,A -85,B 0,C 180,E1 -4215.275,E2 -4215.275} C_VEL
LIN {X 0,Y 532.515,Z 293.409,A -85,B 0,C 180,E1 -4216.623,E2 -4216.623} C_VEL
LIN {X 0,Y 532.295,Z 305.839,A -85,B 0,C 180,E1 -4216.933,E2 -4216.933} C_VEL
LIN {X 0,Y 532.048,Z 318.711,A -85,B 0,C 180,E1 -4217.412,E2 -4217.412} C_VEL
LIN {X 0,Y 531.849,Z 330.246,A -85,B 0,C 180,E1 -4217.995,E2 -4217.995} C_VEL
LIN {X 0,Y 531.557,Z 341.836,A -85,B 0,C 180,E1 -4218.755,E2 -4218.755} C_VEL
LIN {X 0,Y 531.291,Z 352.335,A -85,B 0,C 180,E1 -4219.617,E2 -4219.617} C_VEL
LIN {X 0,Y 531.07,Z 360.916,A -85,B 0,C 180,E1 -4220.479,E2 -4220.479} C_VEL
LIN {X 0,Y 530.901,Z 368.821,A -85,B 0,C 180,E1 -4221.436,E2 -4221.436} C_VEL
LIN {X 0,Y 530.709,Z 376.553,A -85,B 0,C 180,E1 -4222.582,E2 -4222.582} C_VEL
LIN {X 0,Y 530.637,Z 383.646,A -85,B 0,C 180,E1 -4223.918,E2 -4223.918} C_VEL
LIN {X 0,Y 530.459,Z 388.376,A -85,B 0,C 180,E1 -4225.06,E2 -4225.06} C_VEL
LIN {X 0,Y 530.516,Z 391.998,A -85,B 0,C 180,E1 -4226.203,E2 -4226.203} C_VEL
LIN {X 0,Y 530.483,Z 393.872,A -85,B 0,C 180,E1 -4226.963,E2 -4226.963} C_VEL
LIN {X 0,Y 530.412,Z 395.286,A -85,B 0,C 180,E1 -4227.722,E2 -4227.722} C_VEL
LIN {X 0,Y 530.345,Z 396.911,A -85,B 0,C 180,E1 -4229.241,E2 -4229.241} C_VEL
LIN {X 0,Y 530.344,Z 397.15,A -85,B 0,C 180,E1 -4230,E2 -4230} C_VEL
LIN {X 0,Y 530.344,Z 396.967,A -85,B 0,C 180,E1 -4230.76,E2 -4230.76} C_VEL
LIN {X 0,Y 530.413,Z 395.415,A -85,B 0,C 180,E1 -4232.278,E2 -4232.278} C_VEL
LIN {X 0,Y 530.483,Z 394.056,A -85,B 0,C 180,E1 -4233.038,E2 -4233.038} C_VEL
LIN {X 0,Y 530.523,Z 391.184,A -85,B 0,C 180,E1 -4234.179,E2 -4234.179} C_VEL
LIN {X 0,Y 530.524,Z 387.289,A -85,B 0,C 180,E1 -4235.321,E2 -4235.321} C_VEL
LIN {X 0,Y 530.605,Z 381.656,A -85,B 0,C 180,E1 -4236.587,E2 -4236.587} C_VEL
LIN {X 0,Y 530.759,Z 374.717,A -85,B 0,C 180,E1 -4237.801,E2 -4237.801} C_VEL
LIN {X 0,Y 530.926,Z 366.546,A -85,B 0,C 180,E1 -4238.948,E2 -4238.948} C_VEL
LIN {X 0,Y 531.132,Z 358.185,A -85,B 0,C 180,E1 -4239.905,E2 -4239.905} C_VEL
LIN {X 0,Y 531.398,Z 347.867,A -85,B 0,C 180,E1 -4240.863,E2 -4240.863} C_VEL
LIN {X 0,Y 531.654,Z 337.22,A -85,B 0,C 180,E1 -4241.659,E2 -4241.659} C_VEL
LIN {X 0,Y 531.926,Z 326.474,A -85,B 0,C 180,E1 -4242.301,E2 -4242.301} C_VEL
LIN {X 0,Y 532.151,Z 313.938,A -85,B 0,C 180,E1 -4242.877,E2 -4242.877} C_VEL
LIN {X 0,Y 532.344,Z 300.48,A -85,B 0,C 180,E1 -4243.309,E2 -4243.309} C_VEL
LIN {X 0,Y 532.499,Z 287.099,A -85,B 0,C 180,E1 -4243.573,E2 -4243.573} C_VEL
LIN {X 0,Y 532.723,Z 194.745,A -85,B 0,C 180,E1 -4244.825,E2 -4244.825} C_VEL
LIN {X 0,Y 531.262,Z 186.052,A -85,B 0,C 180,E1 -4245.014,E2 -4245.014} C_VEL
LIN {X 0,Y 531.519,Z 170.384,A -85,B 0,C 180,E1 -4247.705,E2 -4247.705} C_VEL
LIN {X 0,Y 531.932,Z 153.443,A -85,B 0,C 180,E1 -4250.706,E2 -4250.706} C_VEL
LIN {X 0,Y 530.985,Z 147.406,A -85,B 0,C 180,E1 -4251.881,E2 -4251.881} C_VEL
LIN {X 0,Y 531.007,Z 147.339,A -85,B 0,C 180,E1 -4255.057,E2 -4255.057} C_VEL
LIN {X 0,Y 531.014,Z 147.337,A -85,B 0,C 180,E1 -4257.595,E2 -4257.595} C_VEL
LIN {X 0,Y 530.975,Z 147.341,A -85,B 0,C 180,E1 -4260.645,E2 -4260.645} C_VEL
LIN {X 0,Y 530.989,Z 147.341,A -85,B 0,C 180,E1 -4263.772,E2 -4263.772} C_VEL
LIN {X 0,Y 530.966,Z 147.346,A -85,B 0,C 180,E1 -4266.557,E2 -4266.557} C_VEL
LIN {X 0,Y 530.975,Z 147.34,A -85,B 0,C 180,E1 -4269.853,E2 -4269.853} C_VEL
LIN {X 0,Y 530.978,Z 147.344,A -85,B 0,C 180,E1 -4272.456,E2 -4272.456} C_VEL
LIN {X 0,Y 530.975,Z 147.34,A -85,B 0,C 180,E1 -4275.621,E2 -4275.621} C_VEL
LIN {X 0,Y 530.996,Z 147.338,A -85,B 0,C 180,E1 -4278.564,E2 -4278.564} C_VEL
LIN {X 0,Y 530.952,Z 147.345,A -85,B 0,C 180,E1 -4281.529,E2 -4281.529} C_VEL
LIN {X 0,Y 530.971,Z 147.331,A -85,B 0,C 180,E1 -4284.381,E2 -4284.381} C_VEL
LIN {X 0,Y 530.962,Z 147.337,A -85,B 0,C 180,E1 -4287.133,E2 -4287.133} C_VEL
LIN {X 0,Y 530.964,Z 147.348,A -85,B 0,C 180,E1 -4289.803,E2 -4289.803} C_VEL
LIN {X 0,Y 531.011,Z 147.334,A -85,B 0,C 180,E1 -4292.466,E2 -4292.466} C_VEL
LIN {X 0,Y 530.982,Z 147.339,A -85,B 0,C 180,E1 -4294.941,E2 -4294.941} C_VEL
LIN {X 0,Y 530.964,Z 147.342,A -85,B 0,C 180,E1 -4298.246,E2 -4298.246} C_VEL
LIN {X 0,Y 530.985,Z 147.338,A -85,B 0,C 180,E1 -4300.677,E2 -4300.677} C_VEL
LIN {X 0,Y 530.979,Z 147.339,A -85,B 0,C 180,E1 -4303.071,E2 -4303.071} C_VEL
LIN {X 0,Y 531.011,Z 147.336,A -85,B 0,C 180,E1 -4305.436,E2 -4305.436} C_VEL
LIN {X 0,Y 531.029,Z 147.332,A -85,B 0,C 180,E1 -4308.549,E2 -4308.549} C_VEL
LIN {X 0,Y 531.048,Z 147.334,A -85,B 0,C 180,E1 -4311.629,E2 -4311.629} C_VEL
LIN {X 0,Y 531.111,Z 147.322,A -85,B 0,C 180,E1 -4314.685,E2 -4314.685} C_VEL
LIN {X 0,Y 531.127,Z 147.324,A -85,B 0,C 180,E1 -4317.725,E2 -4317.725} C_VEL
LIN {X 0,Y 531.144,Z 147.319,A -85,B 0,C 180,E1 -4320.758,E2 -4320.758} C_VEL
LIN {X 0,Y 531.096,Z 147.326,A -85,B 0,C 180,E1 -4323.034,E2 -4323.034} C_VEL
LIN {X 0,Y 531.065,Z 147.328,A -85,B 0,C 180,E1 -4326.077,E2 -4326.077} C_VEL
LIN {X 0,Y 531.012,Z 147.34,A -85,B 0,C 180,E1 -4329.138,E2 -4329.138} C_VEL
LIN {X 0,Y 531.022,Z 147.331,A -85,B 0,C 180,E1 -4332.225,E2 -4332.225} C_VEL
LIN {X 0,Y 530.987,Z 147.346,A -85,B 0,C 180,E1 -4335.35,E2 -4335.35} C_VEL
LIN {X 0,Y 530.977,Z 147.336,A -85,B 0,C 180,E1 -4338.522,E2 -4338.522} C_VEL
LIN {X 0,Y 530.991,Z 147.342,A -85,B 0,C 180,E1 -4340.938,E2 -4340.938} C_VEL
LIN {X 0,Y 530.956,Z 147.339,A -85,B 0,C 180,E1 -4344.226,E2 -4344.226} C_VEL
LIN {X 0,Y 530.994,Z 147.34,A -85,B 0,C 180,E1 -4346.744,E2 -4346.744} C_VEL
LIN {X 0,Y 530.974,Z 147.345,A -85,B 0,C 180,E1 -4349.323,E2 -4349.323} C_VEL
LIN {X 0,Y 530.958,Z 147.342,A -85,B 0,C 180,E1 -4352.1,E2 -4352.1} C_VEL
LIN {X 0,Y 530.963,Z 147.345,A -85,B 0,C 180,E1 -4354.851,E2 -4354.851} C_VEL
LIN {X 0,Y 530.96,Z 147.339,A -85,B 0,C 180,E1 -4357.508,E2 -4357.508} C_VEL
LIN {X 0,Y 530.976,Z 147.341,A -85,B 0,C 180,E1 -4360.434,E2 -4360.434} C_VEL
LIN {X 0,Y 530.929,Z 147.349,A -85,B 0,C 180,E1 -4363.278,E2 -4363.278} C_VEL
LIN {X 0,Y 530.971,Z 147.341,A -85,B 0,C 180,E1 -4365.623,E2 -4365.623} C_VEL
LIN {X 0,Y 530.96,Z 147.346,A -85,B 0,C 180,E1 -4368.562,E2 -4368.562} C_VEL
LIN {X 0,Y 530.953,Z 147.338,A -85,B 0,C 180,E1 -4371.53,E2 -4371.53} C_VEL
LIN {X 0,Y 530.949,Z 147.347,A -85,B 0,C 180,E1 -4374.38,E2 -4374.38} C_VEL
LIN {X 0,Y 530.966,Z 147.346,A -85,B 0,C 180,E1 -4377.134,E2 -4377.134} C_VEL
LIN {X 0,Y 530.953,Z 147.342,A -85,B 0,C 180,E1 -4379.802,E2 -4379.802} C_VEL
LIN {X 0,Y 530.975,Z 147.34,A -85,B 0,C 180,E1 -4382.476,E2 -4382.476} C_VEL
LIN {X 0,Y 530.951,Z 147.347,A -85,B 0,C 180,E1 -4384.94,E2 -4384.94} C_VEL
LIN {X 0,Y 530.988,Z 147.474,A -85,B 0,C 180,E1 -4387.018,E2 -4387.018} C_VEL
LIN {X 0,Y 532.126,Z 154.463,A -85,B 0,C 180,E1 -4388.296,E2 -4388.296} C_VEL
LIN {X 0,Y 531.737,Z 171.167,A -85,B 0,C 180,E1 -4391.106,E2 -4391.106} C_VEL
LIN {X 0,Y 531.368,Z 189.057,A -85,B 0,C 180,E1 -4394.071,E2 -4394.071} C_VEL
LIN {X 0,Y 531.324,Z 195.249,A -85,B 0,C 180,E1 -4395.039,E2 -4395.039} C_VEL
LIN {X 0,Y 532.803,Z 205.136,A -85,B 0,C 180,E1 -4395.235,E2 -4395.235} C_VEL
LIN {X 0,Y 532.44,Z 302.685,A -85,B 0,C 180,E1 -4396.572,E2 -4396.572} C_VEL
LIN {X 0,Y 532.244,Z 315.961,A -85,B 0,C 180,E1 -4396.907,E2 -4396.907} C_VEL
LIN {X 0,Y 531.967,Z 329.24,A -85,B 0,C 180,E1 -4397.409,E2 -4397.409} C_VEL
LIN {X 0,Y 531.767,Z 340.836,A -85,B 0,C 180,E1 -4398.013,E2 -4398.013} C_VEL
LIN {X 0,Y 531.514,Z 351.963,A -85,B 0,C 180,E1 -4398.753,E2 -4398.753} C_VEL
LIN {X 0,Y 531.255,Z 362.386,A -85,B 0,C 180,E1 -4399.616,E2 -4399.616} C_VEL
LIN {X 0,Y 531.056,Z 370.906,A -85,B 0,C 180,E1 -4400.478,E2 -4400.478} C_VEL
LIN {X 0,Y 530.883,Z 378.765,A -85,B 0,C 180,E1 -4401.435,E2 -4401.435} C_VEL
LIN {X 0,Y 530.675,Z 386.437,A -85,B 0,C 180,E1 -4402.581,E2 -4402.581} C_VEL
LIN {X 0,Y 530.603,Z 393.508,A -85,B 0,C 180,E1 -4403.917,E2 -4403.917} C_VEL
LIN {X 0,Y 530.459,Z 398.21,A -85,B 0,C 180,E1 -4405.059,E2 -4405.059} C_VEL
LIN {X 0,Y 530.516,Z 401.803,A -85,B 0,C 180,E1 -4406.202,E2 -4406.202} C_VEL
LIN {X 0,Y 530.457,Z 403.655,A -85,B 0,C 180,E1 -4406.962,E2 -4406.962} C_VEL
LIN {X 0,Y 530.411,Z 405.043,A -85,B 0,C 180,E1 -4407.722,E2 -4407.722} C_VEL
LIN {X 0,Y 530.344,Z 406.639,A -85,B 0,C 180,E1 -4409.24,E2 -4409.24} C_VEL
LIN {X 0,Y 530.343,Z 406.855,A -85,B 0,C 180,E1 -4410,E2 -4410} C_VEL
LIN {X 0,Y 530.361,Z 406.037,A -85,B 0,C 180,E1 -4411.518,E2 -4411.518} C_VEL
LIN {X 0,Y 530.411,Z 405.047,A -85,B 0,C 180,E1 -4412.278,E2 -4412.278} C_VEL
LIN {X 0,Y 530.457,Z 403.66,A -85,B 0,C 180,E1 -4413.037,E2 -4413.037} C_VEL
LIN {X 0,Y 530.522,Z 400.74,A -85,B 0,C 180,E1 -4414.178,E2 -4414.178} C_VEL
LIN {X 0,Y 530.524,Z 396.785,A -85,B 0,C 180,E1 -4415.32,E2 -4415.32} C_VEL
LIN {X 0,Y 530.596,Z 391.102,A -85,B 0,C 180,E1 -4416.579,E2 -4416.579} C_VEL
LIN {X 0,Y 530.729,Z 384.051,A -85,B 0,C 180,E1 -4417.8,E2 -4417.8} C_VEL
LIN {X 0,Y 530.911,Z 375.797,A -85,B 0,C 180,E1 -4418.948,E2 -4418.948} C_VEL
LIN {X 0,Y 531.116,Z 367.335,A -85,B 0,C 180,E1 -4419.905,E2 -4419.905} C_VEL
LIN {X 0,Y 531.393,Z 356.874,A -85,B 0,C 180,E1 -4420.863,E2 -4420.863} C_VEL
LIN {X 0,Y 531.641,Z 345.966,A -85,B 0,C 180,E1 -4421.667,E2 -4421.667} C_VEL
LIN {X 0,Y 531.906,Z 335.172,A -85,B 0,C 180,E1 -4422.301,E2 -4422.301} C_VEL
LIN {X 0,Y 532.125,Z 323.53,A -85,B 0,C 180,E1 -4422.829,E2 -4422.829} C_VEL
LIN {X 0,Y 532.315,Z 311.025,A -85,B 0,C 180,E1 -4423.237,E2 -4423.237} C_VEL
LIN {X 0,Y 532.453,Z 298.378,A -85,B 0,C 180,E1 -4423.5,E2 -4423.5} C_VEL
LIN {X 0,Y 532.724,Z 204.087,A -85,B 0,C 180,E1 -4424.781,E2 -4424.781} C_VEL
LIN {X 0,Y 531.321,Z 195.322,A -85,B 0,C 180,E1 -4424.957,E2 -4424.957} C_VEL
LIN {X 0,Y 531.314,Z 191.446,A -85,B 0,C 180,E1 -4425.536,E2 -4425.536} C_VEL
LIN {X 0,Y 531.695,Z 173.556,A -85,B 0,C 180,E1 -4428.495,E2 -4428.495} C_VEL
LIN {X 0,Y 532.072,Z 155.66,A -85,B 0,C 180,E1 -4431.502,E2 -4431.502} C_VEL
LIN {X 0,Y 531.708,Z 151.11,A -85,B 0,C 180,E1 -4432.294,E2 -4432.294} C_VEL
LIN {X 0,Y 530.988,Z 147.415,A -85,B 0,C 180,E1 -4433.008,E2 -4433.008} C_VEL
LIN {X 0,Y 530.968,Z 147.342,A -85,B 0,C 180,E1 -4435.899,E2 -4435.899} C_VEL
LIN {X 0,Y 530.965,Z 147.341,A -85,B 0,C 180,E1 -4438.456,E2 -4438.456} C_VEL
LIN {X 0,Y 530.948,Z 147.347,A -85,B 0,C 180,E1 -4441.079,E2 -4441.079} C_VEL
LIN {X 0,Y 530.982,Z 147.338,A -85,B 0,C 180,E1 -4443.772,E2 -4443.772} C_VEL
LIN {X 0,Y 530.945,Z 147.345,A -85,B 0,C 180,E1 -4446.558,E2 -4446.558} C_VEL
LIN {X 0,Y 530.98,Z 147.343,A -85,B 0,C 180,E1 -4449.442,E2 -4449.442} C_VEL
LIN {X 0,Y 530.956,Z 147.343,A -85,B 0,C 180,E1 -4452.457,E2 -4452.457} C_VEL
LIN {X 0,Y 530.977,Z 147.342,A -85,B 0,C 180,E1 -4455.452,E2 -4455.452} C_VEL
LIN {X 0,Y 530.984,Z 147.34,A -85,B 0,C 180,E1 -4458.563,E2 -4458.563} C_VEL
LIN {X 0,Y 530.946,Z 147.34,A -85,B 0,C 180,E1 -4461.528,E2 -4461.528} C_VEL
LIN {X 0,Y 530.948,Z 147.336,A -85,B 0,C 180,E1 -4464.379,E2 -4464.379} C_VEL
LIN {X 0,Y 530.956,Z 147.348,A -85,B 0,C 180,E1 -4467.132,E2 -4467.132} C_VEL
LIN {X 0,Y 530.948,Z 147.341,A -85,B 0,C 180,E1 -4469.802,E2 -4469.802} C_VEL
LIN {X 0,Y 531,Z 147.339,A -85,B 0,C 180,E1 -4472.467,E2 -4472.467} C_VEL
LIN {X 0,Y 530.976,Z 147.344,A -85,B 0,C 180,E1 -4474.941,E2 -4474.941} C_VEL
LIN {X 0,Y 530.959,Z 147.343,A -85,B 0,C 180,E1 -4478.246,E2 -4478.246} C_VEL
LIN {X 0,Y 530.982,Z 147.346,A -85,B 0,C 180,E1 -4480.677,E2 -4480.677} C_VEL
LIN {X 0,Y 530.961,Z 147.344,A -85,B 0,C 180,E1 -4483.07,E2 -4483.07} C_VEL
LIN {X 0,Y 531.005,Z 147.336,A -85,B 0,C 180,E1 -4485.435,E2 -4485.435} C_VEL
LIN {X 0,Y 531.041,Z 147.335,A -85,B 0,C 180,E1 -4488.55,E2 -4488.55} C_VEL
LIN {X 0,Y 531.036,Z 147.332,A -85,B 0,C 180,E1 -4491.629,E2 -4491.629} C_VEL
LIN {X 0,Y 531.106,Z 147.326,A -85,B 0,C 180,E1 -4494.685,E2 -4494.685} C_VEL
LIN {X 0,Y 531.12,Z 147.321,A -85,B 0,C 180,E1 -4497.725,E2 -4497.725} C_VEL
LIN {X 0,Y 531.143,Z 147.321,A -85,B 0,C 180,E1 -4500.758,E2 -4500.758} C_VEL
LIN {X 0,Y 531.093,Z 147.324,A -85,B 0,C 180,E1 -4503.034,E2 -4503.034} C_VEL
LIN {X 0,Y 531.06,Z 147.332,A -85,B 0,C 180,E1 -4506.077,E2 -4506.077} C_VEL
LIN {X 0,Y 531.043,Z 147.336,A -85,B 0,C 180,E1 -4508.371,E2 -4508.371} C_VEL
LIN {X 0,Y 531.04,Z 147.331,A -85,B 0,C 180,E1 -4511.674,E2 -4511.674} C_VEL
LIN {X 0,Y 531.018,Z 147.332,A -85,B 0,C 180,E1 -4514.956,E2 -4514.956} C_VEL
LIN {X 0,Y 531.004,Z 147.336,A -85,B 0,C 180,E1 -4517.723,E2 -4517.723} C_VEL
LIN {X 0,Y 530.992,Z 147.336,A -85,B 0,C 180,E1 -4520.938,E2 -4520.938} C_VEL
LIN {X 0,Y 530.969,Z 147.349,A -85,B 0,C 180,E1 -4524.225,E2 -4524.225} C_VEL
LIN {X 0,Y 530.994,Z 147.337,A -85,B 0,C 180,E1 -4526.744,E2 -4526.744} C_VEL
LIN {X 0,Y 530.972,Z 147.339,A -85,B 0,C 180,E1 -4529.323,E2 -4529.323} C_VEL
LIN {X 0,Y 530.955,Z 147.348,A -85,B 0,C 180,E1 -4532.101,E2 -4532.101} C_VEL
LIN {X 0,Y 530.974,Z 147.329,A -85,B 0,C 180,E1 -4534.854,E2 -4534.854} C_VEL
LIN {X 0,Y 530.957,Z 147.34,A -85,B 0,C 180,E1 -4537.509,E2 -4537.509} C_VEL
LIN {X 0,Y 530.976,Z 147.342,A -85,B 0,C 180,E1 -4540.434,E2 -4540.434} C_VEL
LIN {X 0,Y 530.954,Z 147.336,A -85,B 0,C 180,E1 -4543.282,E2 -4543.282} C_VEL
LIN {X 0,Y 530.944,Z 147.339,A -85,B 0,C 180,E1 -4543.585,E2 -4543.585} C_VEL
LIN {X 0,Y 530.273,Z 147.43,A -85,B 0,C 180,E1 -4544.219,E2 -4544.219} C_VEL
LIN {X 0,Y 527.425,Z 147.78,A -85,B 0,C 180,E1 -4545.248,E2 -4545.248} C_VEL
LIN {X 0,Y 525.022,Z 148.088,A -85,B 0,C 180,E1 -4546.076,E2 -4546.076} C_VEL
LIN {X 0,Y 523.992,Z 148.211,A -85,B 0,C 180,E1 -4546.716,E2 -4546.716} C_VEL
LIN {X 0,Y 523.909,Z 148.22,A -85,B 0,C 180,E1 -4546.932,E2 -4546.932} C_VEL
LIN {X 0,Y 523.944,Z 148.216,A -85,B 0,C 180,E1 -4549.922,E2 -4549.922} C_VEL
LIN {X 0,Y 523.906,Z 148.221,A -85,B 0,C 180,E1 -4552.869,E2 -4552.869} C_VEL
LIN {X 0,Y 523.933,Z 148.22,A -85,B 0,C 180,E1 -4555.711,E2 -4555.711} C_VEL
LIN {X 0,Y 523.918,Z 148.217,A -85,B 0,C 180,E1 -4558.457,E2 -4558.457} C_VEL
LIN {X 0,Y 523.933,Z 148.219,A -85,B 0,C 180,E1 -4561.126,E2 -4561.126} C_VEL
LIN {X 0,Y 523.983,Z 148.218,A -85,B 0,C 180,E1 -4563.981,E2 -4563.981} C_VEL
LIN {X 0,Y 523.925,Z 148.222,A -85,B 0,C 180,E1 -4566.271,E2 -4566.271} C_VEL
LIN {X 0,Y 523.979,Z 148.364,A -85,B 0,C 180,E1 -4568.098,E2 -4568.098} C_VEL
LIN {X 0,Y 524.964,Z 154.131,A -85,B 0,C 180,E1 -4569.222,E2 -4569.222} C_VEL
LIN {X 0,Y 524.563,Z 170.469,A -85,B 0,C 180,E1 -4572.156,E2 -4572.156} C_VEL
LIN {X 0,Y 524.265,Z 186.038,A -85,B 0,C 180,E1 -4574.865,E2 -4574.865} C_VEL
LIN {X 0,Y 525.175,Z 191.358,A -85,B 0,C 180,E1 -4575,E2 -4575} C_VEL
LIN {X 0,Y 525.911,Z 196.446,A -85,B 0,C 180,E1 -4575.092,E2 -4575.092} C_VEL
LIN {X 0,Y 525.629,Z 293.503,A -85,B 0,C 180,E1 -4576.444,E2 -4576.444} C_VEL
LIN {X 0,Y 525.404,Z 305.922,A -85,B 0,C 180,E1 -4576.758,E2 -4576.758} C_VEL
LIN {X 0,Y 525.108,Z 318.79,A -85,B 0,C 180,E1 -4577.243,E2 -4577.243} C_VEL
LIN {X 0,Y 524.874,Z 331.024,A -85,B 0,C 180,E1 -4577.876,E2 -4577.876} C_VEL
LIN {X 0,Y 524.596,Z 341.909,A -85,B 0,C 180,E1 -4578.604,E2 -4578.604} C_VEL
LIN {X 0,Y 524.305,Z 352.407,A -85,B 0,C 180,E1 -4579.477,E2 -4579.477} C_VEL
LIN {X 0,Y 524.068,Z 360.987,A -85,B 0,C 180,E1 -4580.35,E2 -4580.35} C_VEL
LIN {X 0,Y 523.873,Z 368.89,A -85,B 0,C 180,E1 -4581.32,E2 -4581.32} C_VEL
LIN {X 0,Y 523.649,Z 376.622,A -85,B 0,C 180,E1 -4582.481,E2 -4582.481} C_VEL
LIN {X 0,Y 523.547,Z 383.714,A -85,B 0,C 180,E1 -4583.836,E2 -4583.836} C_VEL
LIN {X 0,Y 523.384,Z 388.443,A -85,B 0,C 180,E1 -4584.993,E2 -4584.993} C_VEL
LIN {X 0,Y 523.443,Z 392.065,A -85,B 0,C 180,E1 -4586.151,E2 -4586.151} C_VEL
LIN {X 0,Y 523.391,Z 393.938,A -85,B 0,C 180,E1 -4586.921,E2 -4586.921} C_VEL
LIN {X 0,Y 523.337,Z 395.352,A -85,B 0,C 180,E1 -4587.691,E2 -4587.691} C_VEL
LIN {X 0,Y 523.251,Z 396.977,A -85,B 0,C 180,E1 -4589.231,E2 -4589.231} C_VEL
LIN {X 0,Y 523.247,Z 397.215,A -85,B 0,C 180,E1 -4590,E2 -4590} C_VEL
LIN {X 0,Y 523.25,Z 397.032,A -85,B 0,C 180,E1 -4590.77,E2 -4590.77} C_VEL
LIN {X 0,Y 523.337,Z 395.479,A -85,B 0,C 180,E1 -4592.309,E2 -4592.309} C_VEL
LIN {X 0,Y 523.391,Z 394.12,A -85,B 0,C 180,E1 -4593.079,E2 -4593.079} C_VEL
LIN {X 0,Y 523.443,Z 391.247,A -85,B 0,C 180,E1 -4594.235,E2 -4594.235} C_VEL
LIN {X 0,Y 523.464,Z 387.352,A -85,B 0,C 180,E1 -4595.393,E2 -4595.393} C_VEL
LIN {X 0,Y 523.543,Z 382.103,A -85,B 0,C 180,E1 -4596.599,E2 -4596.599} C_VEL
LIN {X 0,Y 523.694,Z 374.778,A -85,B 0,C 180,E1 -4597.907,E2 -4597.907} C_VEL
LIN {X 0,Y 523.9,Z 366.606,A -85,B 0,C 180,E1 -4599.069,E2 -4599.069} C_VEL
LIN {X 0,Y 524.115,Z 358.244,A -85,B 0,C 180,E1 -4600.039,E2 -4600.039} C_VEL
LIN {X 0,Y 524.427,Z 347.925,A -85,B 0,C 180,E1 -4601.009,E2 -4601.009} C_VEL
LIN {X 0,Y 524.718,Z 336.563,A -85,B 0,C 180,E1 -4601.865,E2 -4601.865} C_VEL
LIN {X 0,Y 524.983,Z 326.528,A -85,B 0,C 180,E1 -4602.466,E2 -4602.466} C_VEL
LIN {X 0,Y 525.221,Z 315.206,A -85,B 0,C 180,E1 -4603.001,E2 -4603.001} C_VEL
LIN {X 0,Y 525.44,Z 302.352,A -85,B 0,C 180,E1 -4603.438,E2 -4603.438} C_VEL
LIN {X 0,Y 525.594,Z 288.67,A -85,B 0,C 180,E1 -4603.73,E2 -4603.73} C_VEL
LIN {X 0,Y 525.796,Z 194.86,A -85,B 0,C 180,E1 -4605.024,E2 -4605.024} C_VEL
LIN {X 0,Y 524.249,Z 186.097,A -85,B 0,C 180,E1 -4605.219,E2 -4605.219} C_VEL
LIN {X 0,Y 524.503,Z 172.671,A -85,B 0,C 180,E1 -4607.543,E2 -4607.543} C_VEL
LIN {X 0,Y 524.962,Z 154.843,A -85,B 0,C 180,E1 -4610.738,E2 -4610.738} C_VEL
LIN {X 0,Y 523.954,Z 148.33,A -85,B 0,C 180,E1 -4612.008,E2 -4612.008} C_VEL
LIN {X 0,Y 523.934,Z 148.223,A -85,B 0,C 180,E1 -4614.571,E2 -4614.571} C_VEL
LIN {X 0,Y 523.95,Z 148.217,A -85,B 0,C 180,E1 -4617.133,E2 -4617.133} C_VEL
LIN {X 0,Y 523.943,Z 148.218,A -85,B 0,C 180,E1 -4619.755,E2 -4619.755} C_VEL
LIN {X 0,Y 523.934,Z 148.224,A -85,B 0,C 180,E1 -4622.449,E2 -4622.449} C_VEL
LIN {X 0,Y 523.932,Z 148.213,A -85,B 0,C 180,E1 -4625.225,E2 -4625.225} C_VEL
LIN {X 0,Y 523.914,Z 148.227,A -85,B 0,C 180,E1 -4628.101,E2 -4628.101} C_VEL
LIN {X 0,Y 523.939,Z 148.213,A -85,B 0,C 180,E1 -4631.092,E2 -4631.092} C_VEL
LIN {X 0,Y 523.93,Z 148.223,A -85,B 0,C 180,E1 -4634.228,E2 -4634.228} C_VEL
LIN {X 0,Y 523.903,Z 148.213,A -85,B 0,C 180,E1 -4636.831,E2 -4636.831} C_VEL
LIN {X 0,Y 523.94,Z 148.215,A -85,B 0,C 180,E1 -4638.907,E2 -4638.907} C_VEL
LIN {X 0,Y 523.911,Z 148.227,A -85,B 0,C 180,E1 -4641.898,E2 -4641.898} C_VEL
LIN {X 0,Y 523.927,Z 148.204,A -85,B 0,C 180,E1 -4644.909,E2 -4644.909} C_VEL
LIN {X 0,Y 523.93,Z 148.218,A -85,B 0,C 180,E1 -4647.679,E2 -4647.679} C_VEL
LIN {X 0,Y 523.949,Z 148.215,A -85,B 0,C 180,E1 -4650.676,E2 -4650.676} C_VEL
LIN {X 0,Y 523.947,Z 148.212,A -85,B 0,C 180,E1 -4652.867,E2 -4652.867} C_VEL
LIN {X 0,Y 523.933,Z 148.225,A -85,B 0,C 180,E1 -4655.801,E2 -4655.801} C_VEL
LIN {X 0,Y 523.938,Z 148.213,A -85,B 0,C 180,E1 -4658.766,E2 -4658.766} C_VEL
LIN {X 0,Y 523.942,Z 148.217,A -85,B 0,C 180,E1 -4661.22,E2 -4661.22} C_VEL
LIN {X 0,Y 523.93,Z 148.222,A -85,B 0,C 180,E1 -4663.639,E2 -4663.639} C_VEL
LIN {X 0,Y 523.932,Z 148.221,A -85,B 0,C 180,E1 -4666.028,E2 -4666.028} C_VEL
LIN {X 0,Y 524.005,Z 148.207,A -85,B 0,C 180,E1 -4668.394,E2 -4668.394} C_VEL
LIN {X 0,Y 523.996,Z 148.211,A -85,B 0,C 180,E1 -4671.516,E2 -4671.516} C_VEL
LIN {X 0,Y 524.071,Z 148.199,A -85,B 0,C 180,E1 -4674.614,E2 -4674.614} C_VEL
LIN {X 0,Y 524.099,Z 148.199,A -85,B 0,C 180,E1 -4677.694,E2 -4677.694} C_VEL
LIN {X 0,Y 524.115,Z 148.195,A -85,B 0,C 180,E1 -4680.768,E2 -4680.768} C_VEL
LIN {X 0,Y 524.063,Z 148.203,A -85,B 0,C 180,E1 -4683.075,E2 -4683.075} C_VEL
LIN {X 0,Y 524.027,Z 148.204,A -85,B 0,C 180,E1 -4686.159,E2 -4686.159} C_VEL
LIN {X 0,Y 523.983,Z 148.217,A -85,B 0,C 180,E1 -4689.262,E2 -4689.262} C_VEL
LIN {X 0,Y 523.991,Z 148.211,A -85,B 0,C 180,E1 -4691.737,E2 -4691.737} C_VEL
LIN {X 0,Y 523.985,Z 148.215,A -85,B 0,C 180,E1 -4695.052,E2 -4695.052} C_VEL
LIN {X 0,Y 523.94,Z 148.213,A -85,B 0,C 180,E1 -4697.97,E2 -4697.97} C_VEL
LIN {X 0,Y 523.95,Z 148.215,A -85,B 0,C 180,E1 -4700.411,E2 -4700.411} C_VEL
LIN {X 0,Y 523.903,Z 148.224,A -85,B 0,C 180,E1 -4702.894,E2 -4702.894} C_VEL
LIN {X 0,Y 523.976,Z 148.212,A -85,B 0,C 180,E1 -4706.02,E2 -4706.02} C_VEL
LIN {X 0,Y 523.923,Z 148.222,A -85,B 0,C 180,E1 -4708.876,E2 -4708.876} C_VEL
LIN {X 0,Y 523.913,Z 148.223,A -85,B 0,C 180,E1 -4711.545,E2 -4711.545} C_VEL
LIN {X 0,Y 523.915,Z 148.217,A -85,B 0,C 180,E1 -4714.292,E2 -4714.292} C_VEL
LIN {X 0,Y 523.902,Z 148.218,A -85,B 0,C 180,E1 -4717.133,E2 -4717.133} C_VEL
LIN {X 0,Y 523.934,Z 148.217,A -85,B 0,C 180,E1 -4720.13,E2 -4720.13} C_VEL
LIN {X 0,Y 523.914,Z 148.221,A -85,B 0,C 180,E1 -4722.457,E2 -4722.457} C_VEL
LIN {X 0,Y 523.937,Z 148.22,A -85,B 0,C 180,E1 -4725.311,E2 -4725.311} C_VEL
LIN {X 0,Y 523.921,Z 148.225,A -85,B 0,C 180,E1 -4728.694,E2 -4728.694} C_VEL
LIN {X 0,Y 523.914,Z 148.218,A -85,B 0,C 180,E1 -4731.081,E2 -4731.081} C_VEL
LIN {X 0,Y 523.894,Z 148.223,A -85,B 0,C 180,E1 -4733.825,E2 -4733.825} C_VEL
LIN {X 0,Y 523.94,Z 148.219,A -85,B 0,C 180,E1 -4736.636,E2 -4736.636} C_VEL
LIN {X 0,Y 523.943,Z 148.216,A -85,B 0,C 180,E1 -4739.355,E2 -4739.355} C_VEL
LIN {X 0,Y 523.946,Z 148.217,A -85,B 0,C 180,E1 -4742.288,E2 -4742.288} C_VEL
LIN {X 0,Y 523.903,Z 148.22,A -85,B 0,C 180,E1 -4745.427,E2 -4745.427} C_VEL
LIN {X 0,Y 523.949,Z 148.333,A -85,B 0,C 180,E1 -4746.848,E2 -4746.848} C_VEL
LIN {X 0,Y 525.162,Z 155.596,A -85,B 0,C 180,E1 -4748.2,E2 -4748.2} C_VEL
LIN {X 0,Y 524.767,Z 172.299,A -85,B 0,C 180,E1 -4751.048,E2 -4751.048} C_VEL
LIN {X 0,Y 524.361,Z 190.186,A -85,B 0,C 180,E1 -4754.052,E2 -4754.052} C_VEL
LIN {X 0,Y 524.304,Z 195.032,A -85,B 0,C 180,E1 -4754.823,E2 -4754.823} C_VEL
LIN {X 0,Y 525.601,Z 203.37,A -85,B 0,C 180,E1 -4755.005,E2 -4755.005} C_VEL
LIN {X 0,Y 525.937,Z 208.411,A -85,B 0,C 180,E1 -4755.084,E2 -4755.084} C_VEL
LIN {X 0,Y 525.55,Z 302.621,A -85,B 0,C 180,E1 -4756.392,E2 -4756.392} C_VEL
LIN {X 0,Y 525.343,Z 315.896,A -85,B 0,C 180,E1 -4756.731,E2 -4756.731} C_VEL
LIN {X 0,Y 525.044,Z 329.175,A -85,B 0,C 180,E1 -4757.24,E2 -4757.24} C_VEL
LIN {X 0,Y 524.818,Z 340.596,A -85,B 0,C 180,E1 -4757.841,E2 -4757.841} C_VEL
LIN {X 0,Y 524.552,Z 351.898,A -85,B 0,C 180,E1 -4758.602,E2 -4758.602} C_VEL
